(*		nIndexRange[1].nStartIndex := 0;
		nIndexRange[1].nEndIndex := 1;
		nIndexRange[1].bRangeAccess := TRUE; *)
		stNodeAddInfo.nIndexRangeCount := nIndexRangeCount;
		stNodeAddInfo.stIndexRange := stIndexRange;
		iState	:= iState + 1;
	END_IF

1:	(* open UA session *)
	fbUA_Connect(
		Execute				:= TRUE,
		ServerURL			:= sOpcUA_URL,
		SessionConnectInfo	:= SessionConnectInfo,
		Timeout				:= T#5S,
		ConnectionHdl		=> nConnectionHdl
	);

	IF NOT fbUA_Connect.Busy THEN
		fbUA_Connect(Execute := FALSE);

		IF NOT fbUA_Connect.Error THEN
			(* session open *)
			iState := iState + 1;
		ELSE
			bError			:= TRUE;
			nErrorID		:= fbUA_Connect.ErrorID;
			nConnectionHdl	:= 0;
			iState 			:= 0; (* idle *)
		END_IF
	END_IF


2:	(* GetNS Index *)
	fbUA_GetNamespaceIndex(
		Execute			:= TRUE,
		ConnectionHdl	:= nConnectionHdl,
		NamespaceUri	:= 'PLC1',
		NamespaceIndex	=> nNamespaceIndex
	);

	IF NOT fbUA_GetNamespaceIndex.Busy THEN
		fbUA_GetNamespaceIndex(Execute := FALSE);
		IF NOT fbUA_GetNamespaceIndex.Error THEN
			(* session closed *)
			iState 		:= iState + 1; (* idle *)
		ELSE
			bError		:= TRUE;
			nErrorID	:= fbUA_GetNamespaceIndex.ErrorID;
			iState 		:= 6; (* idle *)
		END_IF
	END_IF


3:	(* Get Node Handle *)
	NodeID.eIdentifierType := eUAIdentifierType_String;
	NodeID.nNamespaceIndex := nNamespaceIndex;
	NodeID.sIdentifier	:= 'invalidArrayDef';
	fbUA_NodeGetHandle(
		Execute			:= TRUE,
		ConnectionHdl	:= nConnectionHdl,
		NodeID			:= NodeID,
		NodeHdl			=> nNodeHdl
	);

	IF NOT fbUA_NodeGetHandle.Busy THEN
		fbUA_NodeGetHandle(Execute := FALSE);

		IF NOT fbUA_NodeGetHandle.Error THEN
			(* session closed *)
			iState 					:= iState + 1; (* idle *)
		ELSE
			bError		:= TRUE;
			nErrorID	:= fbUA_NodeGetHandle.ErrorID;
			iState 		:= 6; (* idle *)
			IF fbUA_NodeGetHandle.ErrorID = 16#E4DD0125 THEN  
				bTestSuccessfull := TRUE;
			END_IF

		END_IF
	END_IF


4: 	(* Should not be reached since gethandle should fail! *)
	iState 		:= iState + 1; 
	bTestSuccessfull := FALSE;
	
5:	(* Release Node Handle *)
	fbUA_NodeReleaseHandle(
		Execute			:= TRUE,
		ConnectionHdl	:= nConnectionHdl,
		NodeHdl			:= nNodeHdl
	);

	IF NOT fbUA_NodeReleaseHandle.Busy THEN
		fbUA_NodeReleaseHandle(Execute := FALSE);

		IF NOT fbUA_NodeReleaseHandle.Error THEN
			(* session closed *)
			iState 		:= iState + 1; (* idle *)
		ELSE
			bError		:= TRUE;
			nErrorID	:= fbUA_NodeReleaseHandle.ErrorID;
			iState 		:= 6; (* idle *)
		END_IF
	END_IF


6:	(* close session *)
	fbUA_Disconnect(
		Execute			:= TRUE,
		ConnectionHdl	:= nConnectionHdl
	);

	IF NOT fbUA_Disconnect.Busy THEN
		fbUA_Disconnect(Execute := FALSE);
		bBusy := FALSE;
		IF NOT fbUA_Disconnect.Error THEN
			(* session closed *)
			iState 		:= 0; (* idle *)
			IF NOT bError THEN 
				bDone 	:= TRUE;
			END_IF
		ELSE
			bError			:= TRUE;
			nErrorID		:= fbUA_Disconnect.ErrorID;
			iState 			:= 0; (* idle *)
			nConnectionHdl	:= 0;
		END_IF
	END_IF
END_CASE

END_PROGRAM

// ---- Tests_Henning/POUs/PRG_READ_List_Henning.TcPOU
PROGRAM PRG_READ_List_Henning
VAR
	fbUA_ConnectEx			: UA_ConnectEx;
	SessionConnectInfoEx	: ST_UASessionConnectInfoEx;
	sOpcUA_URL				: STRING(MAX_STRING_LENGTH);
	nConnectionHdl			: DWORD;

	fbUA_GetNamespaceIndex 	: UA_GetNamespaceIndex;
	nNamespaceIndex			: UINT;
	fbUA_NodeGetHandleList	: UA_NodeGetHandleList;
	fbUA_NodeGetHandle		: UA_NodeGetHandle;
	NodeIDCount				: UINT := 2; 
	NodeIDs					: ARRAY [1..nMaxNodeIDsInList] OF ST_UANodeID;
	NodeID1					: ST_UANodeID; 
	NodeID2					: ST_UANodeID; 
	nNodeHdls				: ARRAY [1..nMaxNodeIDsInList] OF DWORD;

	fbUA_ReadList			: UA_ReadList;
	NodeHdlCount			: UINT := 2; 
	stIndexRange			: ARRAY [1..nMaxIndexRange] OF ST_UAIndexRange;
	nIndexRangeCount		: UINT;
	stNodeAddInfo			: ARRAY [1..nMaxNodeIDsInList] OF ST_UANodeAdditionalInfo;
	stReadListData			: ST_ReadListData; // memory block must contain the Data[], NodeErrorIDs[], TimeStamps[] and cbData_R[]
	cbData					: ARRAY [1..nMaxNodeIDsInList] OF UDINT; (* Bytes to be actually Read *)
	cbData_R				: UDINT;
	cbDataTotal				: UDINT; 
	
	fbUA_NodeReleaseHandleList	: UA_NodeReleaseHandleList;

	fbUA_Disconnect		: UA_Disconnect;

	iState		: INT;
	bTest		: BOOL:= TRUE;  
	bDone		: BOOL;
	bBusy		: BOOL;
	bError		: BOOL;
	nErrorID	: DWORD;
END_VAR


CASE iState OF
0:	(* idle *)
	IF bTest THEN
		bTest		:= FALSE;
		bError		:= FALSE;
		nErrorID	:= 0;

		(* Parameterize *)
		sOpcUA_URL						:= 'opc.tcp://henningm-nb:4842';	(* OpcUA Url of the device with ip address *)

		SessionConnectInfoEx.tConnectTimeout 		:= T#5S;
		SessionConnectInfoEx.tSessionTimeout 		:= T#5S;
		SessionConnectInfoEx.sApplicationName		:= '';
		SessionConnectInfoEx.eSecurityMode 			:= eUASecurityMsgMode_None;
		SessionConnectInfoEx.eSecurityPolicyUri 	:= eUASecurityPolicy_None;
		SessionConnectInfoEx.eTransportProfileUri 	:= eUATransportProfileUri_UATcp;
		SessionConnectInfoEx.stUserIdentTokenType.eUserIdentTokenType  	 := eUAUITT_Anonymous; 
		SessionConnectInfoEx.stUserIdentTokenType.sTokenParam1  		 := 'beckhoff\henningm'; 
		SessionConnectInfoEx.stUserIdentTokenType.sTokenParam2  		 := 'xx'; 
		

(*		nIndexRange[1].nStartIndex := 0;
		nIndexRange[1].nEndIndex := 1;
		nIndexRange[1].bRangeAccess := TRUE; *)
		iState	:= iState + 1;
	END_IF

1:	(* open UA session *)
	fbUA_ConnectEx(
		Execute				:= TRUE,
		ServerURL			:= sOpcUA_URL,
		SessionConnectInfoEx:= SessionConnectInfoEx,
		Timeout				:= T#5S,
		ConnectionHdl		=> nConnectionHdl
	);

	IF NOT fbUA_ConnectEx.Busy THEN
		fbUA_ConnectEx(Execute := FALSE);

		IF NOT fbUA_ConnectEx.Error THEN
			(* session open *)
			iState := iState + 1;
		ELSE
			bError			:= TRUE;
			nErrorID		:= fbUA_ConnectEx.ErrorID;
			nConnectionHdl	:= 0;
			iState 			:= 8; (* idle *)
		END_IF
	END_IF


2:	(* GetNS Index *)
	fbUA_GetNamespaceIndex(
		Execute			:= TRUE,
		ConnectionHdl	:= nConnectionHdl,
		NamespaceUri	:= 'urn:HENNINGM-NB:BeckhoffAutomation:Ua:TpyPLC',
		NamespaceIndex	=> nNamespaceIndex
	);

	IF NOT fbUA_GetNamespaceIndex.Busy THEN
		fbUA_GetNamespaceIndex(Execute := FALSE);
		IF NOT fbUA_GetNamespaceIndex.Error THEN
			(* session closed *)
			iState 		:= iState + 1; (* idle *)
		ELSE
			bError		:= TRUE;
			nErrorID	:= fbUA_GetNamespaceIndex.ErrorID;
			iState 		:= 8; (* idle *)
		END_IF
	END_IF


3:	(* Get Node Handle *)
	NodeID1.eIdentifierType := eUAIdentifierType_String;	(* Get Node Handle *)
	NodeID1.nNamespaceIndex := nNamespaceIndex;
	NodeID1.sIdentifier	:= 'MAIN.iVar1';
	fbUA_NodeGetHandle(
		Execute			:= TRUE,
		ConnectionHdl	:= nConnectionHdl,
		NodeID			:= NodeID1,
		NodeHdl			=> nNodeHdls[1]
	);

	IF NOT fbUA_NodeGetHandle.Busy THEN
		fbUA_NodeGetHandle(Execute := FALSE);

		IF NOT fbUA_NodeGetHandle.Error THEN
			(* node handle received successfully *)
			iState 		:= iState + 1; (* UA_Read *)
		ELSE
			bError		:= TRUE;
			nErrorID	:= fbUA_NodeGetHandle.ErrorID;
			iState 		:= 5; (* release node handle *)
		END_IF
	END_IF;

4:	(* Get Node Handle *)
	NodeID2.eIdentifierType := eUAIdentifierType_String;	(* Get Node Handle *)
	NodeID2.nNamespaceIndex := nNamespaceIndex;
	NodeID2.sIdentifier	:= 'MAIN.iVar2';
	fbUA_NodeGetHandle(
		Execute			:= TRUE,
		ConnectionHdl	:= nConnectionHdl,
		NodeID			:= NodeID2,
		NodeHdl			=> nNodeHdls[2]
	);

	IF NOT fbUA_NodeGetHandle.Busy THEN
		fbUA_NodeGetHandle(Execute := FALSE);

		IF NOT fbUA_NodeGetHandle.Error THEN
			(* node handle received successfully *)
			iState 		:= iState + 1; (* UA_Read *)
		ELSE
			bError		:= TRUE;
			nErrorID	:= fbUA_NodeGetHandle.ErrorID;
			iState 		:= 8; (* release node handle *)
		END_IF
	END_IF;
	
5: 	(* UA_Read *)
	cbData[1] := SIZEOF(stReadListData.nIntVar1);
	cbData[2] := SIZEOF(stReadListData.nIntVar2);
	cbDataTotal := SIZEOF(stReadListData);
	fbUA_ReadList(
		Execute			:= TRUE,
		ConnectionHdl	:= nConnectionHdl,
		NodeHdlCount	:= NodeHdlCount, // 2
		NodeHdls		:= nNodeHdls,
		stNodeAddInfo 	:= stNodeAddInfo,
		pVariable		:= ADR(stReadListData),
		cbData			:= cbData ,
		cbDataTotal		:= cbDataTotal		
		);

	IF NOT fbUA_ReadList.Busy THEN
		fbUA_ReadList( Execute := FALSE, cbData_R => cbData_R);

		IF NOT fbUA_ReadList.Error THEN
			(* session closed *)
			iState 		:= iState + 1; (* idle *)
		ELSE
			bError		:= TRUE;
			nErrorID	:= fbUA_ReadList.ErrorID;
			iState 		:= 8; (* idle *)
		END_IF
	END_IF


6:	(* Release Node Handle *)
	fbUA_NodeReleaseHandleList(
		Execute			:= TRUE,
		ConnectionHdl	:= nConnectionHdl,
		NodeHdlCount	:= NodeHdlCount,
		NodeHdls		:= nNodeHdls
	);

	IF NOT fbUA_NodeReleaseHandleList.Busy THEN
		fbUA_NodeReleaseHandleList(Execute := FALSE);

		IF NOT fbUA_NodeReleaseHandleList.Error THEN
			(* session closed *)
			iState 		:= iState + 1; (* idle *)
		ELSE
			bError		:= TRUE;
			nErrorID	:= fbUA_NodeReleaseHandleList.ErrorID;
			iState 		:= 7; (* idle *)
		END_IF
	END_IF


7:	(* close session *)
	fbUA_Disconnect(
		Execute			:= TRUE,
		ConnectionHdl	:= nConnectionHdl
	);

	IF NOT fbUA_Disconnect.Busy THEN
		fbUA_Disconnect(Execute := FALSE);
		bBusy := FALSE;
		IF NOT fbUA_Disconnect.Error THEN
			(* session closed *)
			iState 		:= 0; (* idle *)
			IF NOT bError THEN 
				bDone 	:= TRUE;
			END_IF
		ELSE
			bError			:= TRUE;
			nErrorID		:= fbUA_Disconnect.ErrorID;
			iState 			:= 0; (* idle *)
			nConnectionHdl	:= 0;
		END_IF
	END_IF
END_CASE

END_PROGRAM

// ---- Test_CloudSample/POUs/ADS/FB_CloudAdsSqlInsert.TcPOU
FUNCTION_BLOCK FB_CloudAdsSqlInsert
VAR_INPUT
	sNetID 			: T_AmsNetID	:='';
	sInsertCmd 		: T_MaxString	:='';
	bExecute		: BOOL;
	tTimeout		: TIME 			:= T#15S;
END_VAR
VAR_OUTPUT
	bBusy 			: BOOL;
	bError 			: BOOL;
	nErrID 			: UDINT;
	sSQLState		: ST_DBSQLError := (sSQLState:='',nSQLErrorCode:=0);
END_VAR
VAR
	RisingEdge		: R_TRIG;
	ReturnCode		: UDINT := 0;
	ReturnValues	: ARRAY [0..15] OF BYTE;
	ADSRDWRITE1		: ADSRDWRT;
	state			: BYTE;
	dummy			: ST_internalSQLError;
END_VAR

RisingEdge(CLK:=bExecute);
IF RisingEdge.Q THEN
	state := 1;
END_IF

CASE state OF
	0:
		;
	1:
		bBusy := TRUE;
		bError := FALSE;
		nErrID := 0;

		ReturnCode := 0;
		sSQLState.sSQLState := '';
		sSQLState.nSQLErrorCode := 0;

		MEMSET(ADR(ReturnValues), 0, SIZEOF(ReturnValues));

		ADSRDWRITE1(WRTRD:= FALSE);
		ADSRDWRITE1(
			NETID:= sNetID,
			PORT:= 21372,
			IDXGRP:= 524290,
			IDXOFFS:= 1,
			WRITELEN:= SIZEOF(sInsertCmd),
			SRCADDR:= ADR(sInsertCmd),
			READLEN:= SIZEOF(ReturnValues),
			DESTADDR:= ADR(ReturnValues),
			WRTRD:= TRUE,
			TMOUT:= tTimeout);
		state := 2;
	2:
		ADSRDWRITE1( WRTRD:=FALSE);
		IF NOT ADSRDWRITE1.BUSY THEN
			state:= 3;
		END_IF
	3:
		bBusy := ADSRDWRITE1.BUSY;
		bError := ADSRDWRITE1.ERR;
		nErrID := ADSRDWRITE1.ERRID;

		MEMCPY(ADR(ReturnCode), ADR(ReturnValues)+12, SIZEOF(ReturnCode));

		IF NOT ADSRDWRITE1.ERR THEN
			 IF ReturnCode <> 0 THEN
				bError 	:= TRUE;
				nErrID 	:= ReturnCode;
				MEMCPY(ADR(dummy), ADR(ReturnValues), SIZEOF(dummy));
				sSQLState.nSQLErrorCode := dummy.nSQLErrorCode;
				sSQLState.sSQLState := dummy.sSQLState;
			ELSE
				sSQLState.sSQLState := '00000';
				sSQLState.nSQLErrorCode := 0;
			END_IF
		END_IF
		state := 0;
END_CASE

END_FUNCTION_BLOCK

// ---- Test_CloudSample/POUs/CloudSample.TcPOU
PROGRAM CloudSample
VAR
	(* Declarations for Cloud connect to Microsoft Azure Cloud *)
	bInsertAzure					: BOOL;
	bInsertAzureCyclic				: BOOL;
	nStateAzure						: BYTE := 0;
	R_TRIGAzure						: R_TRIG;
	
	ObjectNodeID					: ST_UANodeID;
	MethodNodeID					: ST_UANodeID;

	bErrorAzure						: BOOL; 
	nErrorIDAzure					: DWORD;
				
	fb_OpcUAConnectAzure			: UA_Connect;
	SessionConnectInfo				: ST_UASessionConnectInfo;
	sOpcUA_URLAzure					: STRING(MAX_STRING_LENGTH);
	hUAConnectionHdlAzure			: UDINT;
	
	fbUA_OpcUAGetNSIndexAzure 		: UA_GetNamespaceIndex;
	nNamespaceIndexAzure			: UINT;
	nNamespaceIndex					: UINT;
	
	fb_OpcUAMethodGetHandleAzure	: UA_MethodGetHandle;
	hUAMethodHandleAzure			: UDINT;
	
	fb_OpcUAMethodCallAzure			: UA_MethodCall;
	hUAMethodCallAzure				: UDINT;
	nUAMethodCallOutputAzure		: ST_UASQLState;
	stOutputArgInfo					: ARRAY [1..nNumberOfOutputArguments] OF ST_UAMethodArgInfo;
	fbBuildSqlInsertAzure			: FB_BuildSQLInsert;
	sSqlInsertAzure					: STRING(100);	
	stOutputArgInfoAndData			: ST_CloudSampleRes;
	
	fb_OpcUADisconnectAzure			: UA_Disconnect;
	bUADisconnectStartAzure			: BOOL; 
	
(* Method Call Struct *)
	InputArguments				: ARRAY [1..nNumberOfInputArguments] OF ST_UAMethodArgInfo; (*ReadWriteReq has 6 input parameters *)
	OutputArguments				: ARRAY [1..1024] OF BYTE; (* Bytes to be read *)
	nArg						: INT;
	nInputData					: ARRAY [1..nInputArgSize] OF BYTE; // (sNetID(24) + Port(2) + IG(4) + IO(4))
	nOffset						: UDINT;

	
	sNetID						: T_AmsNetId := '127.0.0.1.1.1'; 		(* AmsNetId OF the Target *)
	nPort						: INT; 				(* Port number	*)
	nIndexGroup					: DINT;				(* IndexGroup*)
	nIndexOffset				: DINT; 			(* IndexOffset*)
//	cbWriteData					: UDINT;			(* Count of bytes to be read*)
	bInputDataError				: BOOL; 
	
	(* Miscellaneous variables *)
	fbRandom					: DRAND;
	lrRandom					: LREAL;
	sRandom						: STRING(MAX_DATA_ACCURACY);
	sRandom2					: STRING(MAX_DATA_ACCURACY);
	fbNTGetTime					: NT_GetTime;
	bBusyTime					: BOOL;
	stTime						: TIMESTRUCT;
	
	bInit						: BOOL := TRUE;
END_VAR
VAR CONSTANT
	nInputArgSize				: UDINT := 34;  //(sNetID(24) + Port(2) + IG(4) + IO(4))
	nNumberOfInputArguments 	: UDINT := 6;	
	nNumberOfOutputArguments	: UDINT := 1;		(* 6 *)
	cbReadData					: UDINT := SIZEOF(ST_UASQLState);			(* Count of bytes to be read*)
END_VAR

(* Create random number for upload into the Cloud *)
fbRandom(
	Seed := 1,
	Num => lrRandom);
lrRandom := lrRandom * 10;
sRandom := LREAL_TO_STRING(lrRandom);

(* The value of Poti 1 will be used to write into Cloud *)
sRandom2 := INT_TO_STRING(us_Poti_1);
IF bInit THEN 
	M_Init();
	bInit := FALSE; 
END_IF
R_TRIGAzure(CLK := bInsertAzure);
(* Upload once to Microsoft Azure Cloud *)
CASE nStateAzure OF
	0:
	 	(* To start this sample you have to set a rising edge to the variable bInsertAzure *)
		IF R_TRIGAzure.Q OR bInsertAzureCyclic THEN
			M_Init();
			nStateAzure 	:= 1;		
			bInsertAzure 	:= FALSE;
			bInsertAzureCyclic := TRUE;
			bErrorAzure 	:= FALSE; 
			nErrorIDAzure 	:= 0; 
		END_IF
			
	1:
		(* Get System Time to create timestamp*)
		fbNTGetTime(
			NETID 	:= '',
			START	:= TRUE,
			TMOUT 	:= T#5S,
			BUSY 	=> bBusyTime,
			TIMESTR => stTime);
		
		IF NOT bBusyTime THEN
			fbNTGetTime(START := FALSE);
			nStateAzure := 2;
		END_IF

	2:
		(* Establish session to OPC-UA Server *)
		IF hUAConnectionHdlAzure = 0 THEN
			fb_OpcUAConnectAzure(
				Execute 			:= TRUE,
				ServerUrl 			:= 'opc.tcp://ew2013vm.cloudapp.net:4840',
				SessionConnectInfo 	:= SessionConnectInfo,
				Timeout 			:= T#5S,
				ConnectionHdl 		=> hUAConnectionHdlAzure
				);
		ELSE
			nStateAzure := 4; 		
		END_IF
		
		IF NOT fb_OpcUAConnectAzure.Busy THEN
			fb_OpcUAConnectAzure(Execute := FALSE);
			IF NOT fb_OpcUAConnectAzure.Error THEN
				nStateAzure := 3;
			ELSE
				(* Error Occurred *)
				bErrorAzure	 := TRUE; 
				nErrorIDAzure := fb_OpcUAConnectAzure.ErrorID;
			END_IF	
		END_IF	
		
	3: 
		(* GetNS Index *)
		fbUA_OpcUAGetNSIndexAzure(
			Execute			:= TRUE,
			ConnectionHdl	:= hUAConnectionHdlAzure,
			NamespaceUri	:= 'ADSAMS',
			NamespaceIndex	=> nNamespaceIndexAzure
		);
	
		IF NOT fbUA_OpcUAGetNSIndexAzure.Busy THEN
			fbUA_OpcUAGetNSIndexAzure(Execute := FALSE);
			IF NOT fbUA_OpcUAGetNSIndexAzure.Error THEN
				(* session closed *)
				ObjectNodeID.eIdentifierType := eUAIdentifierType_String;
				ObjectNodeID.nNamespaceIndex := nNamespaceIndexAzure;
				ObjectNodeID.sIdentifier	 := 'ADSAMS';
				
				MethodNodeID.eIdentifierType := eUAIdentifierType_String;
				MethodNodeID.nNamespaceIndex := nNamespaceIndexAzure;
				MethodNodeID.sIdentifier	 := 'ADSAMS.AdsReadWriteReq';
				nStateAzure := 4; (* method *)
			ELSE
				(* Error occurred *)
				bErrorAzure	 := TRUE; 
				nErrorIDAzure := fbUA_OpcUAGetNSIndexAzure.ErrorID;
			END_IF
		END_IF
	
	4:
		(* Get method handle for AdsReadWrite method *)
		IF hUAMethodHandleAzure = 0 THEN
			fb_OpcUAMethodGetHandleAzure(
				Execute 		:= TRUE,
				Timeout 		:= T#15S,
				ConnectionHdl  	:= hUAConnectionHdlAzure,
				ObjectNodeID	:= ObjectNodeID,
				MethodNodeID	:= MethodNodeID,
				MethodHdl 		=> hUAMethodHandleAzure);
		END_IF
		
		IF NOT fb_OpcUAMethodGetHandleAzure.Busy THEN 
			fb_OpcUAMethodGetHandleAzure(Execute := FALSE);
			IF NOT fb_OpcUAMethodGetHandleAzure.Error THEN
				nStateAzure := 5;		
			ELSE
				(* Error occurred *)
				bErrorAzure	  := TRUE; 
				nErrorIDAzure := fb_OpcUAMethodGetHandleAzure.ErrorID;
			END_IF
		END_IF 
	
	5:
		(* Prepare SQL Insert for Cloud *)
		fbBuildSqlInsertAzure(
			sTableName 		:= 'Zaehlerdaten',
			stTimestamp 	:= stTime,
			uiMesstellenID 	:= 2,
			stLogger 		:= 'HelloWorld',
			rMesswert 		:= 42,
			stEinheit 		:= 'Celsius',
			sValue 			:= sRandom2,
			sQuery 			=> sSqlInsertAzure);
		
		(* Write data to the Microsoft Azure cloud via OPC-UA *)
		nNamespaceIndex := nNamespaceIndexAzure;
		M_MethodCallInit();
		stOutputArgInfoAndData.stOutputArgInfo[1].nLenData:= SIZEOF(ST_UASQLState);
		IF bInputDataError = FALSE THEN 
			fb_OpcUAMethodCallAzure(
				Execute					:= TRUE,
				Timeout 				:= T#15S,
				ConnectionHdl			:= hUAConnectionHdlAzure,
				MethodHdl				:= hUAMethodHandleAzure,
				nNumberOfInputArguments := nNumberOfInputArguments,		(* 6 *)
				pInputArgInfo			:= ADR(InputArguments),
				cbInputArgInfo			:= SIZEOF(InputArguments),
				pInputArgData			:= ADR(nInputData),
				cbInputArgData			:= nOffset,
				pInputWriteData			:= ADR(sSqlInsertAzure),
				cbInputWriteData		:= INT_TO_UDINT(LEN(sSqlInsertAzure))+1,
				nNumberOfOutputArguments:= nNumberOfOutputArguments,		(* 6 *)
				pOutputArgInfo			:= ADR(stOutputArgInfo),
				cbOutputArgInfo			:= SIZEOF(stOutputArgInfo),
				pOutputArgInfoAndData	:= ADR(stOutputArgInfoAndData),
				cbOutputArgInfoAndData	:= SIZEOF(stOutputArgInfoAndData)		
			);
			IF NOT fb_OpcUAMethodCallAzure.Busy THEN
				fb_OpcUAMethodCallAzure(Execute := FALSE);
				IF NOT fb_OpcUAMethodCallAzure.Error THEN
					bInsertAzure := FALSE;
					nStateAzure := 0;
					nUAMethodCallOutputAzure.nReturnCode := stOutputArgInfoAndData.stUASQLStateInternal.nReturnCode;
					(* ------------ according to TcDatabase.lib *)
					IF nUaMethodCallOutputAzure.nReturnCode <> 0 THEN 
						bErrorAzure := TRUE;
						nErrorIDAzure := stOutputArgInfoAndData.stUASQLStateInternal.nReturnCode;
						nUAMethodCallOutputAzure.sSQLState		:= stOutputArgInfoAndData.stUASQLStateInternal.sSQLState;
						nUAMethodCallOutputAzure.nSQLErrorCode 	:= stOutputArgInfoAndData.stUASQLStateInternal.nSQLErrorCode;
					ELSE
						nUAMethodCallOutputAzure.sSQLState		:= '00000';	
						nUAMethodCallOutputAzure.nSQLErrorCode 	:= 0;		
					END_IF		
					(* ------------- according to TcDatabase.lib *)
				ELSE
					(* Error Occurred *)
					nStateAzure   := 6; 
					bErrorAzure	  := TRUE; 
					nErrorIDAzure := fb_OpcUAMethodCallAzure.ErrorID;
				END_IF	
			END_IF
		ELSE
			(* ERROR nInputData array is too small for the data *)
			(* see M_MethodCallInit*)
			;
		END_IF
END_CASE

ACTION M_Init:
(* Parameterize *)
SessionConnectInfo.tConnectTimeout 		:= T#1S;
SessionConnectInfo.tSessionTimeout 		:= T#1S;
SessionConnectInfo.sApplicationName		:= '';
SessionConnectInfo.sApplicationUri 		:= '';
SessionConnectInfo.eSecurityMode 		:= eUASecurityMsgMode_None;
SessionConnectInfo.eSecurityPolicyUri 	:= eUASecurityPolicy_None;
SessionConnectInfo.eTransportProfileUri := eUATransportProfileUri_UATcp;
END_ACTION

ACTION M_MethodCallInit:
bInputDataError := FALSE; 
(* Method Call parameters *)
sNetID				:= '127.0.0.1.1.1'; 		(* AmsNetId OF the Target *)
nPort				:= 21372; 					(* Port number *) (* AMSPORT_DATABASESRV := 21372 = 16#537C*)
nIndexGroup			:= 16#80002;				(* IndexGroup*) 
nIndexOffset		:= 2; 						(* IndexOffset = DBID (Configurator)*)
//cbWriteData			:= LEN(sSqlInsertAzure)+1;		
//cbReadData			:= 16;	

nOffset := 0;
MEMSET(ADR(InputArguments),0,SIZEOF(InputArguments));
MEMSET(ADR(nInputData),0,SIZEOF(nInputData));

nArg := 1;
(*sNetID := sAmsNetID;*)	(*****l***** NET ID **********)
InputArguments[nArg].DataType			:= eUAType_String;
InputArguments[nArg].ValueRank			:= -1; 							(* Scalar = -1 or Array *)
InputArguments[nArg].ArrayDimensions[1]	:= 0; 							(* Number of Dimension in case its an array *)
InputArguments[nArg].nLenData			:= INT_TO_UDINT(LEN(sNetId)) + 1;				(* Length if its a STRING *)
IF nOffset + INT_TO_UDINT(LEN(sNetId))+1 > nInputArgSize THEN 
	bInputDataError := TRUE;
	RETURN;
ELSE
	MEMCPY(ADR(nInputData)+nOffset,ADR(sNetId),INT_TO_UDINT(LEN(sNetId))+1);				(* VALUE in BYTES FORM *)
	nOffset := nOffset + INT_TO_UDINT(LEN(sNetId))+1;
END_IF

nArg := nArg + 1;
(* nPort := 851;*)			(********** PORT **********)
InputArguments[nArg].DataType			:= eUAType_Int16;
InputArguments[nArg].ValueRank			:= -1; 						(* Scalar = -1 or Array *)
InputArguments[nArg].ArrayDimensions[1]	:= 0; 						(* Number of Dimension in case its an array *)
InputArguments[nArg].nLenData			:= SIZEOF(nPort);			(* Length if its a STRING *)
IF nOffset + SIZEOF(nPort) > nInputArgSize THEN 
	bInputDataError := TRUE;
	RETURN;
ELSE
	MEMCPY(ADR(nInputData)+nOffset,ADR(nPort),SIZEOF(nPort));			(* VALUE in BYTES FORM *)
	nOffset := nOffset + SIZEOF(nPort);
END_IF

nArg := nArg + 1;
(*nIndexGroup := 16#4020;*)	(********** INDEX GROUP **********)
InputArguments[nArg].DataType			:= eUAType_Int32;
InputArguments[nArg].ValueRank			:= -1; 							(* Scalar = -1 or Array *)
InputArguments[nArg].ArrayDimensions[1]	:= 0; 							(* Number of Dimension in case its an array *)
InputArguments[nArg].nLenData			:= SIZEOF(nIndexGroup);			(* Length if its a STRING *)
IF nOffset + SIZEOF(nIndexGroup) > nInputArgSize THEN 
	bInputDataError := TRUE;
	RETURN;
ELSE
	MEMCPY(ADR(nInputData)+nOffset,ADR(nIndexGroup),SIZEOF(nIndexGroup));		(* VALUE in BYTES FORM *)
	nOffset := nOffset + SIZEOF(nIndexGroup);
END_IF


nArg := nArg + 1;
(*nIndexOffset := 0; *)		(********** INDEX OFFSET **********)
InputArguments[nArg].DataType			:= eUAType_Int32;
InputArguments[nArg].ValueRank			:= -1; 							(* Scalar = -1 or Array *)
InputArguments[nArg].ArrayDimensions[1]	:= 0; 							(* Number of Dimension in case its an array *)
InputArguments[nArg].nLenData			:= SIZEOF(nIndexOffset);		(* Length if its a STRING *)
IF nOffset + SIZEOF(nIndexOffset) > nInputArgSize THEN 
	bInputDataError := TRUE;
	RETURN;
ELSE
	MEMCPY(ADR(nInputData)+nOffset,ADR(nIndexOffset),SIZEOF(nIndexOffset));	(* VALUE in BYTES FORM *)
	nOffset := nOffset + SIZEOF(nIndexOffset);
END_IF

nArg := nArg + 1;
(*Data := 2; *)		(*********** WriteData ***********)
InputArguments[nArg].DataType			:= eUAType_ByteString;
InputArguments[nArg].ValueRank			:= -1; 										(* Scalar = -1 or Array *)
InputArguments[nArg].ArrayDimensions[1]	:= 0; 										(* Number of Dimension in case its an array *)
InputArguments[nArg].nLenData			:= INT_TO_UDINT(LEN(sSqlInsertAzure))+1;	(* Length if its a STRING *)

nArg := nArg + 1;
(*Data := 2; *)		(*********** ReadData size ***********)
InputArguments[nArg].DataType			:= eUAType_UInt32;
InputArguments[nArg].ValueRank			:= -1; 						(* Scalar = -1 or Array *)
InputArguments[nArg].ArrayDimensions[1]	:= 0; 						(* Number of Dimension in case its an array *)
InputArguments[nArg].nLenData			:= SIZEOF(cbReadData);		(* Length if its a STRING *)
END_ACTION

END_PROGRAM

// ---- Tests_Henning/POUs/PRG_ArrayTest.TcPOU
PROGRAM PRG_ArrayTest
VAR
	iState: INT;
END_VAR

CASE iState OF
0:	
	PRG_ArrayTest_Read();
	IF(NOT PRG_ArrayTest_Read.bBusy AND NOT PRG_ArrayTest_Read.bError) THEN
		iState := iState+1;
	END_IF
1:
	PRG_ArrayTest_Write();
	IF(NOT PRG_ArrayTest_Write.bBusy AND NOT PRG_ArrayTest_Write.bError) THEN
		iState := iState+1;
	END_IF
2:
	PRG_ArrayTest_ReadWritten();
	IF(NOT PRG_ArrayTest_ReadWritten.bBusy AND NOT PRG_ArrayTest_ReadWritten.bError) THEN
		iState := iState+1;
	END_IF
END_CASE

END_PROGRAM

// ---- Tests_Henning/POUs/PRG_ArrayTest_Read.TcPOU
PROGRAM PRG_ArrayTest_Read
VAR
	fbUA_Connect: UA_Connect;
	SessionConnectInfo: ST_UASessionConnectInfo;
	nConnectionHdl: DWORD;
	fbUA_GetNamespaceIndex: UA_GetNamespaceIndex;
	nNamespaceIndex: UINT;
	fbUA_NodeGetHandle: UA_NodeGetHandle;
	NodeID: ST_UANodeID;
	nNodeHdl: DWORD;
	fbUA_Read: UA_Read;
	stIndexRange: ARRAY[1..nMaxIndexRange] OF ST_UAIndexRange;
	nIndexRangeCount: UINT;
	stNodeAddInfo: ST_UANodeAdditionalInfo;
	Variable: ARRAY[1..nMaxReadData] OF BYTE;
	///DINT; 		// change the data type according to the variable type to be read
	nReadData: STRING;
	fbUA_NodeReleaseHandle: UA_NodeReleaseHandle;
	fbUA_Disconnect: UA_Disconnect;
	iState: INT;
	bTest: BOOL := TRUE;
	bDone: BOOL;
	bBusy: BOOL;
	bError: BOOL;
	nErrorID: DWORD;
	nLoopVars: UINT;
END_VAR

CASE iState OF
0:	(* idle *)
	IF bTest THEN
		bTest		:= FALSE;
		bError		:= FALSE;
		nErrorID	:= 0;
		bBusy 		:= TRUE; 
		SessionConnectInfo.tConnectTimeout 		:= T#9S;
		SessionConnectInfo.tSessionTimeout 		:= T#9S;
		SessionConnectInfo.sApplicationName		:= '';
		SessionConnectInfo.sApplicationUri 		:= '';
		SessionConnectInfo.eSecurityMode 		:= eUASecurityMsgMode_None;
		SessionConnectInfo.eSecurityPolicyUri 	:= eUASecurityPolicy_None;
		SessionConnectInfo.eTransportProfileUri := eUATransportProfileUri_UATcp;

		stNodeAddInfo.nIndexRangeCount := nIndexRangeCount;
		stNodeAddInfo.stIndexRange := stIndexRange;
		iState	:= iState + 1;
	END_IF

1:	(* open UA session *)
	fbUA_Connect(
		Execute				:= TRUE,
		ServerURL			:= GVL_ScalarTests.sOpcUA_URL,
		SessionConnectInfo	:= SessionConnectInfo,
		Timeout				:= T#10S,
		ConnectionHdl		=> nConnectionHdl
	);

	IF NOT fbUA_Connect.Busy THEN
		fbUA_Connect(Execute := FALSE);

		IF NOT fbUA_Connect.Error THEN
			(* session open *)
			iState := iState + 1;
		ELSE
			bError			:= TRUE;
			nErrorID		:= fbUA_Connect.ErrorID;
			nConnectionHdl	:= 0;
			iState 			:= 0; (* idle *)
		END_IF
	END_IF


2:	(* GetNS Index *)
	fbUA_GetNamespaceIndex(
		Execute			:= TRUE,
		ConnectionHdl	:= nConnectionHdl,
		NamespaceUri	:= GVL_ScalarTests.sNodeIDNamespace,
		NamespaceIndex	=> nNamespaceIndex
	);

	IF NOT fbUA_GetNamespaceIndex.Busy THEN
		fbUA_GetNamespaceIndex(Execute := FALSE);

		IF NOT fbUA_GetNamespaceIndex.Error THEN
			(* session closed *)
			iState 		:= iState + 1; (* idle *)
		ELSE
			bError		:= TRUE;
			nErrorID	:= fbUA_GetNamespaceIndex.ErrorID;
			iState 		:= 6; (* idle *)
		END_IF
	END_IF


3:	(* Get Node Handle *)
	NodeID.eIdentifierType := eUAIdentifierType_String;
	NodeID.nNamespaceIndex := nNamespaceIndex;
	NodeID.sIdentifier	:= GVL_ArrayTests.NodeID_Identifiers[nLoopVars]; // 'GVL_static.stat_BSTR_0';
	fbUA_NodeGetHandle(
		Execute			:= TRUE,
		ConnectionHdl	:= nConnectionHdl,
		NodeID			:= NodeID,
		NodeHdl			=> nNodeHdl
	);

	IF NOT fbUA_NodeGetHandle.Busy THEN
		fbUA_NodeGetHandle(Execute := FALSE);

		IF NOT fbUA_NodeGetHandle.Error THEN
			(* session closed *)
			iState 		:= iState + 1; (* idle *)
		ELSE
			bError		:= TRUE;
			nErrorID	:= fbUA_NodeGetHandle.ErrorID;
			iState 		:= 6; (* idle *)
		END_IF
	END_IF


4: 	(* UA_Read *)
	fbUA_Read(
		Execute			:= TRUE,
		ConnectionHdl	:= nConnectionHdl,
		NodeHdl			:= nNodeHdl,
		stNodeAddInfo 	:= stNodeAddInfo,
		cbData			:= GVL_ArrayTests.NodeID_Sizes[nLoopVars], //SIZEOF(nReadData),
		pVariable		:= ADR(GVL_ArrayTests.NodeID_ReadResults[nLoopVars].nData) //Variable
		);

	IF NOT fbUA_Read.Busy THEN
		fbUA_Read(
			Execute 	:= FALSE);

		IF NOT fbUA_Read.Error THEN
			(* session closed *)
			iState 		:= iState + 1; (* idle *)
			//Do we need this? We simply store in UNION! MEMCPY(ADR(nReadData),ADR(Variable),SIZEOF(nReadData));
		ELSE
			bError		:= TRUE;
			nErrorID	:= fbUA_Read.ErrorID;
			iState 		:= 7; (* idle *)
		END_IF
	END_IF



5:	(* Release Node Handle *)
	fbUA_NodeReleaseHandle(
		Execute			:= TRUE,
		ConnectionHdl	:= nConnectionHdl,
		NodeHdl			:= nNodeHdl
	);

	IF NOT fbUA_NodeReleaseHandle.Busy THEN
		fbUA_NodeReleaseHandle(Execute := FALSE);

		IF NOT fbUA_NodeReleaseHandle.Error THEN
			(* session closed *)
			iState 		:= iState + 1; (* idle *)
		ELSE
			bError		:= TRUE;
			nErrorID	:= fbUA_NodeReleaseHandle.ErrorID;
			iState 		:= 6; (* idle *)
		END_IF
	END_IF


6:	(* close session *)
	fbUA_Disconnect(
		Execute			:= TRUE,
		ConnectionHdl	:= nConnectionHdl
	);

	IF NOT fbUA_Disconnect.Busy THEN
		fbUA_Disconnect(Execute := FALSE);

		IF NOT fbUA_Disconnect.Error THEN
			(* session closed *)
			iState 		:= 0; (* idle *)
			//restart with next var, if existing in array
			IF(nLoopVars < nEndOfNodeIDVars) THEN
				nLoopVars := nLoopVars+1;
				bTest := TRUE;
			ELSE 
				bBusy 		:= FALSE;
				//prepare for next call 
				bTest := TRUE;
				nLoopVars := 0;
			END_IF
		ELSE
			bError			:= TRUE;
			nErrorID		:= fbUA_Disconnect.ErrorID;
			iState 			:= 0; (* idle *)
			nConnectionHdl	:= 0;
		END_IF
	END_IF
END_CASE

END_PROGRAM

// ---- Tests_Henning/POUs/PRG_ArrayTest_Write.TcPOU
PROGRAM PRG_ArrayTest_Write
VAR
	fbUA_Connect: UA_Connect;
	SessionConnectInfo: ST_UASessionConnectInfo;
	sOpcUA_URL: STRING(MAX_STRING_LENGTH);
	nConnectionHdl: DWORD;
	fbUA_GetNamespaceIndex: UA_GetNamespaceIndex;
	sNamespaceUri: STRING(MAX_STRING_LENGTH);
	nNamespaceIndex: UINT;
	fbUA_NodeGetHandle: UA_NodeGetHandle;
	NodeID: ST_UANodeID;
	nNodeHdl: DWORD;
	fbUA_Write: UA_Write;
	stIndexRange: ARRAY[1..nMaxIndexRange] OF ST_UAIndexRange;
	nIndexRangeCount: UINT;
	stNodeAddInfo: ST_UANodeAdditionalInfo;
	/// UDINT := 12312345;		// change according to the type of variable
	nWriteData: STRING := 'Hallo';
	Variable: ARRAY[1..nMaxReadData] OF BYTE;
	cbData: UDINT;
	fbUA_NodeReleaseHandle: UA_NodeReleaseHandle;
	fbUA_Disconnect: UA_Disconnect;
	iState: INT;
	bTest: BOOL := TRUE;
	bDone: BOOL;
	bBusy: BOOL;
	bError: BOOL;
	nErrorID: DWORD;
	nLoopVars: UINT;
END_VAR

CASE iState OF
0:	(* idle *)
	IF bTest THEN
		bTest	:= FALSE;
		bError	:= FALSE;
		nErrorID	:= 0;
		bBusy := TRUE; 

		(* Parameterize 
		GVL_ScalarTests.NodeID_WriteCommands[0].bBool := TRUE; 
		GVL_ScalarTests.NodeID_WriteCommands[1].sString := 'WriteTest'; 
		GVL_ScalarTests.NodeID_WriteCommands[2].bByte := 123; 
		GVL_ScalarTests.NodeID_WriteCommands[3].nInt := 124; 
		GVL_ScalarTests.NodeID_WriteCommands[4].nUdint := 125; 
		GVL_ScalarTests.NodeID_WriteCommands[5].nLReal := 1.23456; //R8x 
		GVL_ScalarTests.NodeID_WriteCommands[6].bByte := 111; 
		GVL_ScalarTests.NodeID_WriteCommands[7].nInt := 112; 
		GVL_ScalarTests.NodeID_WriteCommands[8].nUdint := 113; 
		*)
		
		SessionConnectInfo.tConnectTimeout 		:= T#9S;
		SessionConnectInfo.tSessionTimeout 		:= T#9S;
		SessionConnectInfo.sApplicationName		:= '';
		SessionConnectInfo.sApplicationUri 		:= '';
		SessionConnectInfo.eSecurityMode 		:= eUASecurityMsgMode_None;
		SessionConnectInfo.eSecurityPolicyUri 	:= eUASecurityPolicy_None;
		SessionConnectInfo.eTransportProfileUri := eUATransportProfileUri_UATcp;
		
		stNodeAddInfo.nIndexRangeCount := nIndexRangeCount;
		stNodeAddInfo.stIndexRange := stIndexRange;
		iState	:= iState + 1;
	END_IF

1:	(* open UA session *)
	fbUA_Connect(
		Execute				:= TRUE,
		ServerURL			:= GVL_ScalarTests.sOpcUA_URL,
		SessionConnectInfo	:= SessionConnectInfo,
		Timeout				:= T#10S,
		ConnectionHdl		=> nConnectionHdl
	);

	IF NOT fbUA_Connect.Busy THEN
		fbUA_Connect(Execute := FALSE);

		IF NOT fbUA_Connect.Error THEN
			(* session open *)
			iState := iState + 1;
		ELSE
			bError			:= TRUE;
			nErrorID		:= fbUA_Connect.ErrorID;
			nConnectionHdl	:= 0;
			iState 			:= 0; (* idle *)
		END_IF
	END_IF


2:	(* GetNS Index *)
	fbUA_GetNamespaceIndex(
		Execute			:= TRUE,
		ConnectionHdl	:= nConnectionHdl,
		NamespaceUri	:= GVL_ScalarTests.sNodeIDNamespace,
		NamespaceIndex	=> nNamespaceIndex
	);

	IF NOT fbUA_GetNamespaceIndex.Busy THEN
		fbUA_GetNamespaceIndex(Execute := FALSE);

		IF NOT fbUA_GetNamespaceIndex.Error THEN
			(* session closed *)
			iState 		:= iState + 1; (* idle *)
		ELSE
			bError		:= TRUE;
			nErrorID	:= fbUA_GetNamespaceIndex.ErrorID;
			iState 		:= 6; (* idle *)
		END_IF
	END_IF


3:	(* Get Node Handle *)
	NodeID.eIdentifierType := eUAIdentifierType_String;
	NodeID.nNamespaceIndex := nNamespaceIndex;
	NodeID.sIdentifier	:= GVL_ArrayTests.NodeID_Identifiers[nLoopVars]; // 'GVL_static.stat_BSTR_0';
	fbUA_NodeGetHandle(
		Execute			:= TRUE,
		ConnectionHdl	:= nConnectionHdl,
		NodeID			:= NodeID,
		NodeHdl			=> nNodeHdl
	);

	IF NOT fbUA_NodeGetHandle.Busy THEN
		fbUA_NodeGetHandle(Execute := FALSE);

		IF NOT fbUA_NodeGetHandle.Error THEN
			(* session closed *)
			IF SIZEOF(nWriteData) <= nMaxReadData THEN 
				iState 		:= iState + 1; (* idle *)
				MEMSET(ADR(Variable),0,SIZEOF(Variable));
				MEMCPY(ADR(Variable),ADR(nWriteData),SIZEOF(nWriteData));
			ELSE
				//cannot write buffer too small -> increase the value of nMaxData in GVL
				bError		:= TRUE;
				iState 		:= 6; (* idle *)
			END_IF
		ELSE
			bError		:= TRUE;
			nErrorID	:= fbUA_NodeGetHandle.ErrorID;
			iState 		:= 6; (* idle *)
		END_IF
	END_IF


4: 	(* UA_Write *)
	fbUA_Write(
		Execute			:= TRUE,
		ConnectionHdl	:= nConnectionHdl,
		NodeHdl			:= nNodeHdl,
		stNodeAddInfo	:= stNodeAddInfo,
		cbData			:= GVL_ArrayTests.NodeID_Sizes[nLoopVars], //SIZEOF(nWriteData),
		pVariable		:= ADR(GVL_ArrayTests.NodeID_WriteCommands[nLoopVars].nData) // Variable		:= Variable
		);

	IF NOT fbUA_Write.Busy THEN
		fbUA_Write(
			Execute 		:= FALSE);

		IF NOT fbUA_Write.Error THEN
			(* session closed *)
			iState 		:= iState + 1; (* idle *)
		ELSE
			bError		:= TRUE;
			nErrorID	:= fbUA_Write.ErrorID;
			iState 		:= 7; (* idle *)
		END_IF
	END_IF


5:	(* Release Node Handle *)
	fbUA_NodeReleaseHandle(
		Execute			:= TRUE,
		ConnectionHdl	:= nConnectionHdl,
		NodeHdl			:= nNodeHdl
	);

	IF NOT fbUA_NodeReleaseHandle.Busy THEN
		fbUA_NodeReleaseHandle(Execute := FALSE);

		IF NOT fbUA_NodeReleaseHandle.Error THEN
			(* session closed *)
			iState 		:= iState + 1; (* idle *)
		ELSE
			bError		:= TRUE;
			nErrorID	:= fbUA_NodeReleaseHandle.ErrorID;
			iState 		:= 6; (* idle *)
		END_IF
	END_IF


6:	(* close session *)
	fbUA_Disconnect(
		Execute			:= TRUE,
		ConnectionHdl	:= nConnectionHdl
	);

	IF NOT fbUA_Disconnect.Busy THEN
		fbUA_Disconnect(Execute := FALSE);

		IF NOT fbUA_Disconnect.Error THEN
			(* session closed *)
			iState 		:= 0; (* idle *)			//restart with next var, if existing in array
			IF(nLoopVars < nEndOfNodeIDVars) THEN
				nLoopVars := nLoopVars+1;
				bTest := TRUE;
			ELSE 
				bBusy 		:= FALSE;
				//prepare for next call 
				nLoopVars := 0;
			END_IF
		ELSE
			bError		:= TRUE;
			nErrorID	:= fbUA_Disconnect.ErrorID;
			iState 		:= 0; (* idle *)
			nConnectionHdl	:= 0;
		END_IF
	END_IF
END_CASE

END_PROGRAM

// ---- Tests_Henning/POUs/PRG_ArrayTest_ReadWritten.TcPOU
PROGRAM PRG_ArrayTest_ReadWritten
VAR
	fbUA_Connect: UA_Connect;
	SessionConnectInfo: ST_UASessionConnectInfo;
	nConnectionHdl: DWORD;
	fbUA_GetNamespaceIndex: UA_GetNamespaceIndex;
	nNamespaceIndex: UINT;
	fbUA_NodeGetHandle: UA_NodeGetHandle;
	NodeID: ST_UANodeID;
	nNodeHdl: DWORD;
	fbUA_Read: UA_Read;
	stIndexRange: ARRAY[1..nMaxIndexRange] OF ST_UAIndexRange;
	nIndexRangeCount: UINT;
	stNodeAddInfo: ST_UANodeAdditionalInfo;
	Variable: ARRAY[1..nMaxReadData] OF BYTE;
	///DINT; 		// change the data type according to the variable type to be read
	nReadData: STRING;
	fbUA_NodeReleaseHandle: UA_NodeReleaseHandle;
	fbUA_Disconnect: UA_Disconnect;
	iState: INT;
	bTest: BOOL := TRUE;
	bDone: BOOL;
	bBusy: BOOL;
	bError: BOOL;
	nErrorID: DWORD;
	nLoopVars: UINT;
	counter: UDINT;
	a: ARRAY[1..nMaxReadDataArray] OF BYTE;
	b: ARRAY[1..nMaxReadDataArray] OF BYTE;
	a_: BYTE;
	b_: BYTE;
	nTmpL: UINT;
END_VAR

CASE iState OF
0:	(* idle *)
	IF bTest THEN
		bTest		:= FALSE;
		bError		:= FALSE;
		nErrorID	:= 0;
		bBusy 		:= TRUE; 
		SessionConnectInfo.tConnectTimeout 		:= T#9S;
		SessionConnectInfo.tSessionTimeout 		:= T#9S;
		SessionConnectInfo.sApplicationName		:= '';
		SessionConnectInfo.sApplicationUri 		:= '';
		SessionConnectInfo.eSecurityMode 		:= eUASecurityMsgMode_None;
		SessionConnectInfo.eSecurityPolicyUri 	:= eUASecurityPolicy_None;
		SessionConnectInfo.eTransportProfileUri := eUATransportProfileUri_UATcp;

		stNodeAddInfo.nIndexRangeCount := nIndexRangeCount;
		stNodeAddInfo.stIndexRange := stIndexRange;
		iState	:= iState + 1;
	END_IF

1:	(* open UA session *)
	fbUA_Connect(
		Execute				:= TRUE,
		ServerURL			:= GVL_ScalarTests.sOpcUA_URL,
		SessionConnectInfo	:= SessionConnectInfo,
		Timeout				:= T#10S,
		ConnectionHdl		=> nConnectionHdl
	);

	IF NOT fbUA_Connect.Busy THEN
		fbUA_Connect(Execute := FALSE);

		IF NOT fbUA_Connect.Error THEN
			(* session open *)
			iState := iState + 1;
		ELSE
			bError			:= TRUE;
			nErrorID		:= fbUA_Connect.ErrorID;
			nConnectionHdl	:= 0;
			iState 			:= 0; (* idle *)
		END_IF
	END_IF


2:	(* GetNS Index *)
	fbUA_GetNamespaceIndex(
		Execute			:= TRUE,
		ConnectionHdl	:= nConnectionHdl,
		NamespaceUri	:= GVL_ScalarTests.sNodeIDNamespace,
		NamespaceIndex	=> nNamespaceIndex
	);

	IF NOT fbUA_GetNamespaceIndex.Busy THEN
		fbUA_GetNamespaceIndex(Execute := FALSE);

		IF NOT fbUA_GetNamespaceIndex.Error THEN
			(* session closed *)
			iState 		:= iState + 1; (* idle *)
		ELSE
			bError		:= TRUE;
			nErrorID	:= fbUA_GetNamespaceIndex.ErrorID;
			iState 		:= 6; (* idle *)
		END_IF
	END_IF


3:	(* Get Node Handle *)
	NodeID.eIdentifierType := eUAIdentifierType_String;
	NodeID.nNamespaceIndex := nNamespaceIndex;
	NodeID.sIdentifier	:= GVL_ArrayTests.NodeID_Identifiers[nLoopVars]; // 'GVL_static.stat_BSTR_0';
	fbUA_NodeGetHandle(
		Execute			:= TRUE,
		ConnectionHdl	:= nConnectionHdl,
		NodeID			:= NodeID,
		NodeHdl			=> nNodeHdl
	);

	IF NOT fbUA_NodeGetHandle.Busy THEN
		fbUA_NodeGetHandle(Execute := FALSE);

		IF NOT fbUA_NodeGetHandle.Error THEN
			(* session closed *)
			iState 		:= iState + 1; (* idle *)
		ELSE
			bError		:= TRUE;
			nErrorID	:= fbUA_NodeGetHandle.ErrorID;
			iState 		:= 6; (* idle *)
		END_IF
	END_IF


4: 	(* UA_Read *)
	fbUA_Read(
		Execute			:= TRUE,
		ConnectionHdl	:= nConnectionHdl,
		NodeHdl			:= nNodeHdl,
		stNodeAddInfo 	:= stNodeAddInfo,
		cbData			:= GVL_ArrayTests.NodeID_Sizes[nLoopVars], //SIZEOF(nReadData),		
		pVariable		:= ADR(GVL_ArrayTests.NodeID_ReadWrittenResults[nLoopVars].nData) //Variable
		);

	IF NOT fbUA_Read.Busy THEN
		fbUA_Read(
			Execute 	:= FALSE);

		IF NOT fbUA_Read.Error THEN
			(* session closed *)
			iState 		:= iState + 1; (* idle *)
			a := GVL_ArrayTests.NodeID_WriteCommands[nLoopVars].nData;
			b := GVL_ArrayTests.NodeID_ReadWrittenResults[nLoopVars].nData;
			FOR counter:=1 TO fbUA_Read.cbData_R //fbUA_Read.GVL_ScalarTests.NodeID_Sizes[nLoopVars]
			DO
				a_ := a[counter];
				b_ := b[counter];
				IF(NOT a_ = b_) THEN
					EXIT;
				END_IF
			END_FOR
			IF(Counter = fbUA_Read.cbData_R+1) THEN //GVL_ScalarTests.NodeID_Sizes[nLoopVars]+1) THEN //all bytes are equal as long as length site is defined
				GVL_ArrayTests.NodeID_CheckReadWrite[nLoopVars] := TRUE;
			END_IF 
			//Do we need this? We simply store in UNION! MEMCPY(ADR(nReadData),ADR(Variable),SIZEOF(nReadData));
		ELSE
			bError		:= TRUE;
			nErrorID	:= fbUA_Read.ErrorID;
			iState 		:= 7; (* idle *)
		END_IF
	END_IF



5:	(* Release Node Handle *)
	fbUA_NodeReleaseHandle(
		Execute			:= TRUE,
		ConnectionHdl	:= nConnectionHdl,
		NodeHdl			:= nNodeHdl
	);

	IF NOT fbUA_NodeReleaseHandle.Busy THEN
		fbUA_NodeReleaseHandle(Execute := FALSE);

		IF NOT fbUA_NodeReleaseHandle.Error THEN
			(* session closed *)
			iState 		:= iState + 1; (* idle *)
		ELSE
			bError		:= TRUE;
			nErrorID	:= fbUA_NodeReleaseHandle.ErrorID;
			iState 		:= 6; (* idle *)
		END_IF
	END_IF


6:	(* close session *)
	fbUA_Disconnect(
		Execute			:= TRUE,
		ConnectionHdl	:= nConnectionHdl
	);

	IF NOT fbUA_Disconnect.Busy THEN
		fbUA_Disconnect(Execute := FALSE);

		IF NOT fbUA_Disconnect.Error THEN
			(* session closed *)
			iState 		:= 0; (* idle *)
			//restart with next var, if existing in array
			IF(nLoopVars < nEndOfNodeIDVars) THEN
				nLoopVars := nLoopVars+1;
				bTest := TRUE;
			ELSE 
				bBusy 		:= FALSE;
				//prepare for next call 
				bTest := TRUE;
				nLoopVars := 0;
			END_IF
		ELSE
			bError			:= TRUE;
			nErrorID		:= fbUA_Disconnect.ErrorID;
			iState 			:= 0; (* idle *)
			nConnectionHdl	:= 0;
		END_IF
	END_IF
END_CASE

END_PROGRAM

// ---- Tests_Henning/POUs/PRG_CallInOut1DimParam.TcPOU
PROGRAM PRG_CallInOut1DimParam
VAR
	///CallInOutMultiParams(numberIn1(uInt32),numberIn2(UInt32),numberOut1(UInt32),numberOut2(UINT32));
	fbUA_Connect		: UA_Connect;
	SessionConnectInfo	: ST_UASessionConnectInfo;
	sOpcUA_URL			: STRING(MAX_STRING_LENGTH);
	nConnectionHdl		: DWORD;
	
	fbUA_GetNamespaceIndex	: UA_GetNamespaceIndex;
	nNamespaceIndex			: UINT;
	
	fbUA_MethodGetHandle: UA_MethodGetHandle;
	nMethodHdl			: DWORD;
	ObjectNodeID		: ST_UANodeID;
	MethodNodeID		: ST_UANodeID;
	fbUA_MethodCall		: UA_MethodCall;
	InputArguments		: ARRAY[1..nNumberOfInputArguments] OF ST_UAMethodArgInfo;
	nInputData			: ARRAY[1..nInputArgSize] OF BYTE;
	stOutputArgInfoAndData	: ST_UAMethodCall_CallInOut1DimParam;
	stOutputArgInfo		: ARRAY[1..nNumberOfOutputArguments] OF ST_UAMethodArgInfo;
	numberIn1			: UDINT;
	numberIn2			: UDINT;
	
	fbUA_MethodReleaseHandle	: UA_MethodReleaseHandle;
	
	fbUA_Disconnect	: UA_Disconnect;
	
	/// Count of bytes to be written 
	cbWriteData		: UDINT;
	
	nArg			: INT;
	nOffset			: UDINT;
	bInputDataError	: BOOL;
	bTest			: BOOL := TRUE;
	bDone			: BOOL;
	bBusy			: BOOL;
	bError			: BOOL;
	nErrorID		: DWORD;
	iState			: INT;
	
END_VAR
VAR CONSTANT
	nNumberOfInputArguments	: UDINT := 1;
	nNumberOfOutputArguments: UDINT := 1;
	nInputArgSize			: UDINT := 8; 
END_VAR

(*
CallInOut1DimParams(	[numberIn1(uInt32),	numberIn2(UInt32)]
						[numberOut1(UInt32),numberOut2(UINT32),	numberOut3(UINT32)]
);
*)

CASE iState OF

0:	(* idle *)
	IF bTest THEN
		bTest		:= FALSE;
		bError		:= FALSE;
		nErrorID	:= 0;
		stOutputArgInfoAndData.output1 	:= 0; 
		stOutputArgInfoAndData.output2 	:= 0; 
		stOutputArgInfoAndData.output3 	:= 0; 
		(* Parameterize *)
		sOpcUA_URL		:= 'opc.tcp://localhost:4841';	(* OpcUA Url of the device with ip address *)

		SessionConnectInfo.tConnectTimeout 		:= T#9M;
		SessionConnectInfo.tSessionTimeout 		:= T#9M;
		SessionConnectInfo.sApplicationName		:= '';
		SessionConnectInfo.sApplicationUri 		:= '';
		SessionConnectInfo.eSecurityMode 		:= eUASecurityMsgMode_None;
		SessionConnectInfo.eSecurityPolicyUri 	:= eUASecurityPolicy_None;
		SessionConnectInfo.eTransportProfileUri := eUATransportProfileUri_UATcp;

		iState	:= iState + 1;
	END_IF

1:	(* open UA session *)
	fbUA_Connect(
		Execute				:= TRUE,
		ServerURL			:= sOpcUA_URL,
		SessionConnectInfo	:= SessionConnectInfo,
		Timeout				:= T#10S,
		ConnectionHdl		=> nConnectionHdl
	);

	IF NOT fbUA_Connect.Busy THEN
		fbUA_Connect(Execute := FALSE);

		IF NOT fbUA_Connect.Error THEN
			(* connected *)
			iState := iState + 1;
		ELSE
			bError			:= TRUE;
			nErrorID		:= fbUA_Connect.ErrorID;
			nConnectionHdl	:= 0;
			iState 			:= 0; (* idle *)
		END_IF
	END_IF


2:	(* GetNS Index *)
	fbUA_GetNamespaceIndex(
		Execute			:= TRUE,
		ConnectionHdl	:= nConnectionHdl,
		NamespaceUri	:= 'PLC1',
		NamespaceIndex	=> nNamespaceIndex
	);

	IF NOT fbUA_GetNamespaceIndex.Busy THEN
		fbUA_GetNamespaceIndex(Execute := FALSE);

		IF NOT fbUA_GetNamespaceIndex.Error THEN
			(* namespace index read successfully *)
			iState 		:= iState + 1; (* get node handle *)
		ELSE
			bError		:= TRUE;
			nErrorID	:= fbUA_GetNamespaceIndex.ErrorID;
			iState 		:= 7; (* disconnect *)
		END_IF
	END_IF

3:	(* Get Method Handle *)
		ObjectNodeID.eIdentifierType := eUAIdentifierType_String;
		ObjectNodeID.nNamespaceIndex := nNamespaceIndex;
		ObjectNodeID.sIdentifier	:= 'TestMethods';
	
		MethodNodeID.eIdentifierType := eUAIdentifierType_String;
		MethodNodeID.nNamespaceIndex := nNamespaceIndex;
		MethodNodeID.sIdentifier	:= 'TestMethods.CallInOut1DimParam';

		M_Init();
		IF bInputDataError = FALSE THEN
			iState 	:= iState + 1;
		ELSE
			bBusy		:= FALSE; 
			bError 		:= TRUE;
			nErrorID 	:= 16#70A; //out of memory
		END_IF


4:	(* Method Get Handle *)
	fbUA_MethodGetHandle(
			Execute			:= TRUE,
			ConnectionHdl	:= nConnectionHdl,
			ObjectNodeID	:= ObjectNodeID,
			MethodNodeID 	:= MethodNodeID,
			MethodHdl		=> nMethodHdl
		);
	IF NOT fbUA_MethodGetHandle.Busy THEN
		fbUA_MethodGetHandle(Execute := FALSE);

		IF NOT fbUA_MethodGetHandle.Error THEN
			(*  *)
			iState := iState + 1; (* Call Method *)
		ELSE
			bError		:= TRUE;
			nErrorID	:= fbUA_MethodGetHandle.ErrorID;
			iState	 	:= 6; (* Release method Handle *)
		END_IF
	END_IF


5:	(* Method Call *)
	fbUA_MethodCall(
		Execute					:= TRUE,
		Timeout					:= T#20S,
		ConnectionHdl			:= nConnectionHdl,
		MethodHdl				:= nMethodHdl,
		nNumberOfInputArguments := nNumberOfInputArguments, 
		pInputArgData			:= ADR(nInputData),
		cbInputArgData			:= cbWriteData,
		pInputArgInfo			:= ADR(InputArguments),
		cbInputArgInfo			:= SIZEOF(InputArguments),
		nNumberOfOutputArguments:= nNumberOfOutputArguments,
		pOutputArgInfo			:= ADR(stOutputArgInfo),
		cbOutputArgInfo			:= SIZEOF(stOutputArgInfo),
		pOutputArgInfoAndData	:= ADR(stOutputArgInfoAndData),
		cbOutputArgInfoAndData	:= SIZEOF(stOutputArgInfoAndData)	
	);
	IF NOT fbUA_MethodCall.Busy THEN
		fbUA_MethodCall(Execute := FALSE);
		IF NOT fbUA_MethodCall.Error THEN
			(*  *)
			iState 	:= iState + 1; (* Release handle *)
		ELSE
			bError		:= TRUE;
			nErrorID	:= fbUA_MethodCall.ErrorID;
			iState		:= 6; (* Release method handle *)
		END_IF
	END_IF


6:	(* Release Method Handle *)
	fbUA_MethodReleaseHandle(
		Execute			:= TRUE,
		ConnectionHdl	:= nConnectionHdl,
		MethodHdl		:= nMethodHdl
	);

	IF NOT fbUA_MethodReleaseHandle.Busy THEN
		fbUA_MethodReleaseHandle(Execute := FALSE);
		bBusy := FALSE;
		IF NOT fbUA_MethodReleaseHandle.Error THEN
			(* session closed *)
			iState 	:= 7; (* Disconnect *)
		ELSE
			bError		:= TRUE;
			nErrorID	:= fbUA_MethodReleaseHandle.ErrorID;
			iState 		:= 7; (* Disconnect *)
		END_IF
	END_IF
	
7:	(* Disconnect *) 
	fbUA_Disconnect(
		Execute			:= TRUE,
		ConnectionHdl	:= nConnectionHdl
	);

	IF NOT fbUA_Disconnect.Busy THEN
		fbUA_Disconnect(Execute := FALSE);

		IF NOT fbUA_Disconnect.Error THEN
			(* disconnected *)
			iState 	:= 0; (* idle *)
			bDone 	:= TRUE;
			bBusy 	:= FALSE;
		ELSE
			bBusy 			:= FALSE;
			bError			:= TRUE;
			nErrorID		:= fbUA_Disconnect.ErrorID;
			iState 			:= 0; (* idle *)
			nConnectionHdl	:= 0;
		END_IF
	END_IF
END_CASE

ACTION M_Init:
bInputDataError := FALSE; 
nOffset := 0;
MEMSET(ADR(InputArguments),0,SIZEOF(InputArguments));
MEMSET(ADR(nInputData),0,SIZEOF(nInputData));

nArg := 1;
(*numberIn1*)			(********** Input parameter 1 **********)
InputArguments[nArg].DataType			:= eUAType_UInt32;
InputArguments[nArg].ValueRank			:= 1; 							(* Scalar = -1 or 1Dim-Array =1*)
InputArguments[nArg].ArrayDimensions[1]	:= 2; 							(* Number of Dimension in case its an array *)
InputArguments[nArg].nLenData			:= SIZEOF(numberIn1)+SIZEOF(numberIn2);			(* Length if its a STRING *)

IF nOffset + SIZEOF(numberIn1)+SIZEOF(numberIn2) > nInputArgSize THEN 
	bInputDataError := TRUE;
	RETURN;
ELSE
	MEMCPY(ADR(nInputData)+nOffset,ADR(numberIn1),SIZEOF(numberIn1));				(* VALUE in BYTES FORM *)
	nOffset := nOffset + SIZEOF(numberIn1);
	MEMCPY(ADR(nInputData)+nOffset,ADR(numberIn2),SIZEOF(numberIn2));				(* VALUE in BYTES FORM *)
	nOffset := nOffset + SIZEOF(numberIn2);
END_IF
cbWriteData := nOffset;

//************** Prepare Output Argument information ***********
stOutputArgInfo[1].nLenData := 	SIZEOF(stOutputArgInfoAndData.output1) +
								SIZEOF(stOutputArgInfoAndData.output2) +
								SIZEOF(stOutputArgInfoAndData.output3);
END_ACTION

END_PROGRAM

// ---- Tests_Henning/POUs/PRG_CallInOut1DimStringParam.TcPOU
PROGRAM PRG_CallInOut1DimStringParam
VAR
	///CallInOutMultiParams(numberIn1(uInt32),numberIn2(UInt32),numberOut1(UInt32),numberOut2(UINT32));
	//sIn1: STRING := 'Hallooooo';
	//sIn2: STRING := 'test';
	fbUA_Connect		: UA_Connect;
	SessionConnectInfo	: ST_UASessionConnectInfo;
	sOpcUA_URL			: STRING(MAX_STRING_LENGTH);
	nConnectionHdl		: DWORD;
	
	fbUA_GetNamespaceIndex	: UA_GetNamespaceIndex;
	nNamespaceIndex			: UINT;
	
	fbUA_MethodGetHandle: UA_MethodGetHandle;
	nMethodHdl			: DWORD;
	ObjectNodeID		: ST_UANodeID;
	MethodNodeID		: ST_UANodeID;
	
	fbUA_MethodCall		: UA_MethodCall;
	InputArguments		: ARRAY[1..nNumberOfInputArguments] OF ST_UAMethodArgInfo;
	sInArray			: ARRAY[1..2] OF STRING := ['Halloooo', 'test'] ;
	stOutputArgInfoAndData	: ST_UAMethodCall_CallInOut1DimStringParam;
	nInputData			: ARRAY[1..nInputArgSize] OF BYTE;
	stOutputArgInfo 	: ARRAY[1..nNumberOfOutputArguments] OF ST_UAMethodArgInfo;
	
	fbUA_MethodReleaseHandle: UA_MethodReleaseHandle;
	
	fbUA_Disconnect			: UA_Disconnect;
	
	/// Count of bytes to be written 
	cbWriteData			: UDINT;
	
	nOffset			: UDINT;
	nArg			: INT;
	bInputDataError	: BOOL;
	bTest			: BOOL := TRUE;
	bDone			: BOOL;
	bBusy			: BOOL;
	bError			: BOOL;
	nErrorID		: DWORD;
	iState			: INT;
END_VAR
VAR CONSTANT
	nNumberOfInputArguments	: UDINT := 1;
	nNumberOfOutputArguments: UDINT := 1;
	nInputArgSize			: UDINT := 162;
END_VAR

(*
CallInOut1DimParams(	[numberIn1(uInt32),	numberIn2(UInt32)]
						[numberOut1(UInt32),numberOut2(UINT32),	numberOut3(UINT32)]
);
*)

CASE iState OF

0:	(* idle *)
	IF bTest THEN
		bTest		:= FALSE;
		bError		:= FALSE;
		nErrorID	:= 0;
		stOutputArgInfoAndData.sOutArray[1] 	:= ''; 
		stOutputArgInfoAndData.sOutArray[2] 	:= ''; 
		stOutputArgInfoAndData.sOutArray[3] 	:= ''; 
		(* Parameterize *)
		sOpcUA_URL		:= 'opc.tcp://localhost:4841';	(* OpcUA Url of the device with ip address *)

		SessionConnectInfo.tConnectTimeout 		:= T#9M;
		SessionConnectInfo.tSessionTimeout 		:= T#9M;
		SessionConnectInfo.sApplicationName		:= '';
		SessionConnectInfo.sApplicationUri 		:= '';
		SessionConnectInfo.eSecurityMode 		:= eUASecurityMsgMode_None;
		SessionConnectInfo.eSecurityPolicyUri 	:= eUASecurityPolicy_None;
		SessionConnectInfo.eTransportProfileUri := eUATransportProfileUri_UATcp;

		iState	:= iState + 1;
	END_IF

1:	(* open UA session *)
	fbUA_Connect(
		Execute				:= TRUE,
		ServerURL			:= sOpcUA_URL,
		SessionConnectInfo	:= SessionConnectInfo,
		Timeout				:= T#10S,
		ConnectionHdl		=> nConnectionHdl
	);

	IF NOT fbUA_Connect.Busy THEN
		fbUA_Connect(Execute := FALSE);

		IF NOT fbUA_Connect.Error THEN
			(* connected *)
			iState := iState + 1;
		ELSE
			bError			:= TRUE;
			nErrorID		:= fbUA_Connect.ErrorID;
			nConnectionHdl	:= 0;
			iState 			:= 0; (* idle *)
		END_IF
	END_IF


2:	(* GetNS Index *)
	fbUA_GetNamespaceIndex(
		Execute			:= TRUE,
		ConnectionHdl	:= nConnectionHdl,
		NamespaceUri	:= 'PLC1',
		NamespaceIndex	=> nNamespaceIndex
	);

	IF NOT fbUA_GetNamespaceIndex.Busy THEN
		fbUA_GetNamespaceIndex(Execute := FALSE);

		IF NOT fbUA_GetNamespaceIndex.Error THEN
			(* namespace index read successfully *)
			iState 		:= iState + 1; (* get node handle *)
		ELSE
			bError		:= TRUE;
			nErrorID	:= fbUA_GetNamespaceIndex.ErrorID;
			iState 		:= 7; (* disconnect *)
		END_IF
	END_IF

3:	(* Get Method Handle *)
		ObjectNodeID.eIdentifierType := eUAIdentifierType_String;
		ObjectNodeID.nNamespaceIndex := nNamespaceIndex;
		ObjectNodeID.sIdentifier	:= 'TestMethods';
	
		MethodNodeID.eIdentifierType := eUAIdentifierType_String;
		MethodNodeID.nNamespaceIndex := nNamespaceIndex;
		MethodNodeID.sIdentifier	:= 'TestMethods.CallInOut1DimStringParam';

		M_Init();
		IF bInputDataError = FALSE THEN
			iState 	:= iState + 1;
		ELSE
			bBusy		:= FALSE; 
			bError 		:= TRUE;
			nErrorID 	:= 16#70A; //out of memory
		END_IF


4:	(* Method Get Handle *)
	fbUA_MethodGetHandle(
			Execute			:= TRUE,
			ConnectionHdl	:= nConnectionHdl,
			ObjectNodeID	:= ObjectNodeID,
			MethodNodeID 	:= MethodNodeID,
			MethodHdl		=> nMethodHdl
		);
	IF NOT fbUA_MethodGetHandle.Busy THEN
		fbUA_MethodGetHandle(Execute := FALSE);

		IF NOT fbUA_MethodGetHandle.Error THEN
			(*  *)
			iState := iState + 1; (* Call Method *)
		ELSE
			bError		:= TRUE;
			nErrorID	:= fbUA_MethodGetHandle.ErrorID;
			iState	 	:= 6; (* Release method Handle *)
		END_IF
	END_IF


5:	(* Method Call *)
	fbUA_MethodCall(
		Execute					:= TRUE,
		Timeout					:= T#20S,
		ConnectionHdl			:= nConnectionHdl,
		MethodHdl				:= nMethodHdl,
		nNumberOfInputArguments := nNumberOfInputArguments,		(* 1*)
		pInputArgData			:= ADR(nInputData),
		cbInputArgData			:= cbWriteData,
		pInputArgInfo			:= ADR(InputArguments),
		cbInputArgInfo			:= SIZEOF(InputArguments),
		nNumberOfOutputArguments:= nNumberOfOutputArguments,
		pOutputArgInfo			:= ADR(stOutputArgInfo),
		cbOutputArgInfo			:= SIZEOF(stOutputArgInfo),
		pOutputArgInfoAndData	:= ADR(stOutputArgInfoAndData),
		cbOutputArgInfoAndData	:= SIZEOF(stOutputArgInfoAndData)
	);
	IF NOT fbUA_MethodCall.Busy THEN
		fbUA_MethodCall(Execute := FALSE);

		IF NOT fbUA_MethodCall.Error THEN
			(*  *)
			iState 	:= iState + 1; (* Release handle *)
		ELSE
			bError		:= TRUE;
			nErrorID	:= fbUA_MethodCall.ErrorID;
			iState		:= 6; (* Release method handle *)
		END_IF
	END_IF


6:	(* Release Method Handle *)
	fbUA_MethodReleaseHandle(
		Execute			:= TRUE,
		ConnectionHdl	:= nConnectionHdl,
		MethodHdl		:= nMethodHdl
	);

	IF NOT fbUA_MethodReleaseHandle.Busy THEN
		fbUA_MethodReleaseHandle(Execute := FALSE);
		bBusy := FALSE;
		IF NOT fbUA_MethodReleaseHandle.Error THEN
			(* session closed *)
			iState 	:= 7; (* Disconnect *)
		ELSE
			bError		:= TRUE;
			nErrorID	:= fbUA_MethodReleaseHandle.ErrorID;
			iState 		:= 7; (* Disconnect *)
		END_IF
	END_IF
	
7:	(* Disconnect *) 
	fbUA_Disconnect(
		Execute			:= TRUE,
		ConnectionHdl	:= nConnectionHdl
	);

	IF NOT fbUA_Disconnect.Busy THEN
		fbUA_Disconnect(Execute := FALSE);

		IF NOT fbUA_Disconnect.Error THEN
			(* disconnected *)
			iState 			:= 0; (* idle *)
			bDone 	:= TRUE;
			bBusy 	:= FALSE;
		ELSE
			bBusy 	:= FALSE;
			bError			:= TRUE;
			nErrorID		:= fbUA_Disconnect.ErrorID;
			iState 			:= 0; (* idle *)
			nConnectionHdl	:= 0;
		END_IF
	END_IF
END_CASE

ACTION M_Init:
bInputDataError := FALSE; 
nOffset := 0;
MEMSET(ADR(InputArguments),0,SIZEOF(InputArguments));
MEMSET(ADR(nInputData),0,SIZEOF(nInputData));

nArg := 1;
(*numberIn1*)			(********** Input parameter 1 **********)
InputArguments[nArg].DataType			:= eUAType_String;
InputArguments[nArg].ValueRank			:= 1; 							(* Scalar = -1 or 1Dim-Array =1*)
InputArguments[nArg].ArrayDimensions[1]	:= 2; 							(* Number of Dimension in case its an array *)
InputArguments[nArg].nLenData			:= SIZEOF(sInArray);			(* Length if its a STRING *)
IF nOffset + SIZEOF(sInArray) > nInputArgSize THEN 
	bInputDataError := TRUE;
	RETURN;
ELSE
	MEMCPY(ADR(nInputData)+nOffset,ADR(sInArray),SIZEOF(sInArray));			(* VALUE in BYTES FORM *)
	nOffset := nOffset + SIZEOF(sInArray);
END_IF
//InputArguments[nArg].nLenData			:= SIZEOF(sIn1)+SIZEOF(sIn2);			(* Length if its a STRING *)
//MEMCPY(ADR(nInputData)+nOffset,ADR(sIn1),SIZEOF(sIn1));				(* VALUE in BYTES FORM *)
//nOffset := nOffset + SIZEOF(sIn1);
//MEMCPY(ADR(nInputData)+nOffset,ADR(sIn2),SIZEOF(sIn2));				(* VALUE in BYTES FORM *)
//nOffset := nOffset + SIZEOF(sIn2);

cbWriteData := nOffset;

// ************* Prepare Output variable info **************
stOutputArgInfo[1].nLenData := SIZEOF(stOutputArgInfoAndData.sOutArray);
END_ACTION

END_PROGRAM

// ---- Tests_Henning/POUs/PRG_CallInOutMultiParam.TcPOU
PROGRAM PRG_CallInOutMultiParam
VAR
	///CallInOutMultiParams(numberIn1(uInt32),numberIn2(UInt32),numberOut1(UInt32),numberOut2(UINT32));
	fbUA_Connect			: UA_Connect;
	SessionConnectInfo		: ST_UASessionConnectInfo;
	sOpcUA_URL				: STRING(MAX_STRING_LENGTH);
	nConnectionHdl			: DWORD;
	
	fbUA_GetNamespaceIndex	: UA_GetNamespaceIndex;
	nNamespaceIndex			: UINT;

	fbUA_MethodGetHandle: UA_MethodGetHandle;
	nMethodHdl			: DWORD;
	ObjectNodeID		: ST_UANodeID;
	MethodNodeID		: ST_UANodeID;
	
	fbUA_MethodCall		: UA_MethodCall;
	InputArguments		: ARRAY[1..nNumberOfInputArguments] OF ST_UAMethodArgInfo;
	nInputData			: ARRAY[1..nInputArgSize] OF BYTE;
	OutputArgAndData	: ST_UAMethodCall_CallInOutParam;
	stOutputArgInfo		: ARRAY [1..nNumberOfOutputArguments] OF ST_UAMethodArgInfo;
	
	numberIn1		: UDINT;
	numberIn2		: UDINT;
		
	fbUA_MethodReleaseHandle	: UA_MethodReleaseHandle;
	
	fbUA_Disconnect	: UA_Disconnect;
	
	nArg			: INT;
	cbWriteData		: UDINT;
	nOffset			: UDINT;
	bInputDataError	: BOOL;
	
	bTest		: BOOL := TRUE;
	bDone		: BOOL;
	bBusy		: BOOL;
	bError		: BOOL;
	nErrorID	: DWORD;
	iState		: INT;
END_VAR
VAR CONSTANT
	nNumberOfInputArguments	: UDINT := 2;
	nNumberOfOutputArguments: UDINT := 2; 
	nInputArgSize			: UDINT := 8; 
END_VAR

(*
CallInOutMultiParams(	numberIn1(uInt32),
						numberIn2(UInt32),
						numberOut1(UInt32),
						numberOut2(UINT32)	);
*)

CASE iState OF

0:	(* idle *)
	IF bTest THEN
		bTest		:= FALSE;
		bError		:= FALSE;
		nErrorID	:= 0;
		OutputArgAndData.output1 	:= 0; 
		OutputArgAndData.output2 	:= 0; 
		(* Parameterize *)
		sOpcUA_URL		:= 'opc.tcp://localhost:4841';	(* OpcUA Url of the device with ip address *)

		SessionConnectInfo.tConnectTimeout 		:= T#9S;
		SessionConnectInfo.tSessionTimeout 		:= T#9S;
		SessionConnectInfo.sApplicationName		:= '';
		SessionConnectInfo.sApplicationUri 		:= '';
		SessionConnectInfo.eSecurityMode 		:= eUASecurityMsgMode_None;
		SessionConnectInfo.eSecurityPolicyUri 	:= eUASecurityPolicy_None;
		SessionConnectInfo.eTransportProfileUri := eUATransportProfileUri_UATcp;

		iState	:= iState + 1;
	END_IF

1:	(* open UA session *)
	fbUA_Connect(
		Execute				:= TRUE,
		ServerURL			:= sOpcUA_URL,
		SessionConnectInfo	:= SessionConnectInfo,
		Timeout				:= T#10S,
		ConnectionHdl		=> nConnectionHdl
	);

	IF NOT fbUA_Connect.Busy THEN
		fbUA_Connect(Execute := FALSE);

		IF NOT fbUA_Connect.Error THEN
			(* connected *)
			iState := iState + 1;
		ELSE
			bError			:= TRUE;
			nErrorID		:= fbUA_Connect.ErrorID;
			nConnectionHdl	:= 0;
			iState 			:= 0; (* idle *)
		END_IF
	END_IF


2:	(* GetNS Index *)
	fbUA_GetNamespaceIndex(
		Execute			:= TRUE,
		ConnectionHdl	:= nConnectionHdl,
		NamespaceUri	:= 'PLC1',
		NamespaceIndex	=> nNamespaceIndex
	);

	IF NOT fbUA_GetNamespaceIndex.Busy THEN
		fbUA_GetNamespaceIndex(Execute := FALSE);

		IF NOT fbUA_GetNamespaceIndex.Error THEN
			(* namespace index read successfully *)
			iState 		:= iState + 1; (* get node handle *)
		ELSE
			bError		:= TRUE;
			nErrorID	:= fbUA_GetNamespaceIndex.ErrorID;
			iState 		:= 7; (* disconnect *)
		END_IF
	END_IF

3:	(* Get Method Handle *)
		ObjectNodeID.eIdentifierType := eUAIdentifierType_String;
		ObjectNodeID.nNamespaceIndex := nNamespaceIndex;
		ObjectNodeID.sIdentifier	:= 'TestMethods';
	
		MethodNodeID.eIdentifierType := eUAIdentifierType_String;
		MethodNodeID.nNamespaceIndex := nNamespaceIndex;
		MethodNodeID.sIdentifier	:= 'TestMethods.CallInOutMultiParams';

		M_Init();
		IF bInputDataError = FALSE THEN
			iState 	:= iState + 1;
		ELSE
			bBusy		:= FALSE; 
			bError 		:= TRUE;
			nErrorID 	:= 16#70A; //out of memory
		END_IF


4:	(* Method Get Handle *)
	fbUA_MethodGetHandle(
			Execute			:= TRUE,
			ConnectionHdl	:= nConnectionHdl,
			ObjectNodeID	:= ObjectNodeID,
			MethodNodeID 	:= MethodNodeID,
			MethodHdl		=> nMethodHdl
		);
	IF NOT fbUA_MethodGetHandle.Busy THEN
		fbUA_MethodGetHandle(Execute := FALSE);

		IF NOT fbUA_MethodGetHandle.Error THEN
			(*  *)
			iState := iState + 1; (* Call Method *)
		ELSE
			bError		:= TRUE;
			nErrorID	:= fbUA_MethodGetHandle.ErrorID;
			iState	 	:= 6; (* Release method Handle *)
		END_IF
	END_IF


5:	(* Method Call *)	
	fbUA_MethodCall(
		Execute					:= TRUE,
		Timeout					:= T#20S,
		ConnectionHdl			:= nConnectionHdl,
		MethodHdl				:= nMethodHdl,
		nNumberOfInputArguments := nNumberOfInputArguments,		(* 2 *)
		pInputArgData			:= ADR(nInputData),
		cbInputArgData			:= cbWriteData,
		pInputArgInfo			:= ADR(InputArguments),
		cbInputArgInfo			:= SIZEOF(InputArguments),
		nNumberOfOutputArguments:= nNumberOfOutputArguments,		(* 2 *)
		pOutputArgInfo 			:= ADR(stOutputArgInfo),
		cbOutputArgInfo			:= SIZEOF(stOutputArgInfo),
		pOutputArgInfoAndData	:= ADR(OutputArgAndData),
		cbOutputArgInfoAndData	:= SIZEOF(OutputArgAndData)
	);
	IF NOT fbUA_MethodCall.Busy THEN
		fbUA_MethodCall(Execute := FALSE);

		IF NOT fbUA_MethodCall.Error THEN
			(*  *)
			iState 	:= iState + 1; (* Release handle *)
			//MEMCPY(ADR(OutputArgAndData.output1),ADR(OutputArguments),SIZEOF(OutputArgAndData.output1));
			//MEMCPY(ADR(OutputArgAndData.output2),ADR(OutputArguments)+SIZEOF(OutputArgAndData.output1),SIZEOF(OutputArgAndData.output2));
		ELSE
			bError		:= TRUE;
			nErrorID	:= fbUA_MethodCall.ErrorID;
			iState		:= 6; (* Release method handle *)
		END_IF
	END_IF


6:	(* Release Method Handle *)
	fbUA_MethodReleaseHandle(
		Execute			:= TRUE,
		ConnectionHdl	:= nConnectionHdl,
		MethodHdl		:= nMethodHdl
	);

	IF NOT fbUA_MethodReleaseHandle.Busy THEN
		fbUA_MethodReleaseHandle(Execute := FALSE);
		bBusy := FALSE;
		IF NOT fbUA_MethodReleaseHandle.Error THEN
			(* session closed *)
			iState 	:= 7; (* Disconnect *)
		ELSE
			bError		:= TRUE;
			nErrorID	:= fbUA_MethodReleaseHandle.ErrorID;
			iState 		:= 7; (* Disconnect *)
		END_IF
	END_IF
	
7:	(* Disconnect *) 
	fbUA_Disconnect(
		Execute			:= TRUE,
		ConnectionHdl	:= nConnectionHdl
	);

	IF NOT fbUA_Disconnect.Busy THEN
		fbUA_Disconnect(Execute := FALSE);

		IF NOT fbUA_Disconnect.Error THEN
			(* disconnected *)
			iState 			:= 0; (* idle *)
			bDone 	:= TRUE;
			bBusy 	:= FALSE;
		ELSE
			bBusy 	:= FALSE;
			bError			:= TRUE;
			nErrorID		:= fbUA_Disconnect.ErrorID;
			iState 			:= 0; (* idle *)
			nConnectionHdl	:= 0;
		END_IF
	END_IF
END_CASE

ACTION M_Init:
bInputDataError := FALSE; 
nOffset := 0;
MEMSET(ADR(InputArguments),0,SIZEOF(InputArguments));
MEMSET(ADR(nInputData),0,SIZEOF(nInputData));

nArg := 1;
(*numberIn1*)			(********** Input parameter 1 **********)
InputArguments[nArg].DataType			:= eUAType_UInt32;
InputArguments[nArg].ValueRank			:= -1; 							(* Scalar = -1 or Array *)
InputArguments[nArg].ArrayDimensions[1]	:= 0; 							(* Number of Dimension in case its an array *)
InputArguments[nArg].nLenData			:= SIZEOF(numberIn1);			(* Length if its a STRING *)
IF nOffset + SIZEOF(numberIn1) > nInputArgSize THEN 
	bInputDataError := TRUE;
	RETURN;
ELSE
	MEMCPY(ADR(nInputData)+nOffset,ADR(numberIn1),SIZEOF(numberIn1));				(* VALUE in BYTES FORM *)
	nOffset := nOffset + SIZEOF(numberIn1);
END_IF

cbWriteData := nOffset;
nArg := nArg + 1;
(* numberIn2;*)			(********** Input parameter 2 **********)
InputArguments[nArg].DataType			:= eUAType_UInt32;
InputArguments[nArg].ValueRank			:= -1; 							(* Scalar = -1 or Array *)
InputArguments[nArg].ArrayDimensions[1]	:= 0; 							(* Number of Dimension in case its an array *)
InputArguments[nArg].nLenData			:= SIZEOF(numberIn2);				(* Length if its a STRING *)
IF nOffset + SIZEOF(numberIn2) > nInputArgSize THEN 
	bInputDataError := TRUE;
	RETURN;
ELSE
	MEMCPY(ADR(nInputData)+nOffset,ADR(numberIn2),SIZEOF(numberIn2));				(* VALUE in BYTES FORM *)
	nOffset := nOffset + SIZEOF(numberIn2);
END_IF

cbWriteData := nOffset;

// ************* Prepare Output variable info **************
stOutputArgInfo[1].nLenData := SIZEOF(OutputArgAndData.output1);
stOutputArgInfo[2].nLenData := SIZEOF(OutputArgAndData.output2);
END_ACTION

END_PROGRAM

// ---- Tests_Henning/POUs/PRG_ScalarTest.TcPOU
PROGRAM PRG_ScalarTest
VAR
	iState: INT;
END_VAR

CASE iState OF
0:	
	PRG_ScalarTest_Read();
	IF(NOT PRG_ScalarTest_Read.bBusy AND NOT PRG_ScalarTest_Read.bError) THEN
		iState := iState+1;
		//Reset thus could be reused
		//PRG_ScalarTest_Read.nLoopVars := 0;
		//PRG_ScalarTest_Read.nLoopVars := 0;
	END_IF
1:
	PRG_ScalarTest_Write();
	IF(NOT PRG_ScalarTest_Write.bBusy AND NOT PRG_ScalarTest_Write.bError) THEN
		iState := iState+1;
	END_IF
2:
	PRG_ScalarTest_ReadWritten();
	IF(NOT PRG_ScalarTest_ReadWritten.bBusy AND NOT PRG_ScalarTest_ReadWritten.bError) THEN
		iState := iState+1;
	END_IF
END_CASE

END_PROGRAM

// ---- Tests_Henning/POUs/PRG_ScalarTest_Read.TcPOU
PROGRAM PRG_ScalarTest_Read
VAR
	fbUA_Connect: UA_Connect;
	SessionConnectInfo: ST_UASessionConnectInfo;
	nConnectionHdl: DWORD;
	fbUA_GetNamespaceIndex: UA_GetNamespaceIndex;
	nNamespaceIndex: UINT;
	fbUA_NodeGetHandle: UA_NodeGetHandle;
	NodeID: ST_UANodeID;
	nNodeHdl: DWORD;
	fbUA_Read: UA_Read;
	stIndexRange: ARRAY[1..nMaxIndexRange] OF ST_UAIndexRange;
	nIndexRangeCount: UINT;
	stNodeAddInfo: ST_UANodeAdditionalInfo;
	Variable: ARRAY[1..nMaxReadData] OF BYTE;
	///DINT; 		// change the data type according to the variable type to be read
	nReadData: STRING;
	fbUA_NodeReleaseHandle: UA_NodeReleaseHandle;
	fbUA_Disconnect: UA_Disconnect;
	iState: INT;
	bTest: BOOL := TRUE;
	bDone: BOOL;
	bBusy: BOOL;
	bError: BOOL;
	nErrorID: DWORD;
	nLoopVars: UINT;
END_VAR

CASE iState OF
0:	(* idle *)
	IF bTest THEN
		bTest		:= FALSE;
		bError		:= FALSE;
		nErrorID	:= 0;
		bBusy 		:= TRUE; 
		SessionConnectInfo.tConnectTimeout 		:= T#9S;
		SessionConnectInfo.tSessionTimeout 		:= T#9S;
		SessionConnectInfo.sApplicationName		:= '';
		SessionConnectInfo.sApplicationUri 		:= '';
		SessionConnectInfo.eSecurityMode 		:= eUASecurityMsgMode_None;
		SessionConnectInfo.eSecurityPolicyUri 	:= eUASecurityPolicy_None;
		SessionConnectInfo.eTransportProfileUri := eUATransportProfileUri_UATcp;

		stNodeAddInfo.nIndexRangeCount := nIndexRangeCount;
		stNodeAddInfo.stIndexRange := stIndexRange;
		iState	:= iState + 1;
	END_IF

1:	(* open UA session *)
	fbUA_Connect(
		Execute				:= TRUE,
		ServerURL			:= GVL_ScalarTests.sOpcUA_URL,
		SessionConnectInfo	:= SessionConnectInfo,
		Timeout				:= T#10S,
		ConnectionHdl		=> nConnectionHdl
	);

	IF NOT fbUA_Connect.Busy THEN
		fbUA_Connect(Execute := FALSE);

		IF NOT fbUA_Connect.Error THEN
			(* session open *)
			iState := iState + 1;
		ELSE
			bError			:= TRUE;
			nErrorID		:= fbUA_Connect.ErrorID;
			nConnectionHdl	:= 0;
			iState 			:= 0; (* idle *)
		END_IF
	END_IF


2:	(* GetNS Index *)
	fbUA_GetNamespaceIndex(
		Execute			:= TRUE,
		ConnectionHdl	:= nConnectionHdl,
		NamespaceUri	:= GVL_ScalarTests.sNodeIDNamespace,
		NamespaceIndex	=> nNamespaceIndex
	);

	IF NOT fbUA_GetNamespaceIndex.Busy THEN
		fbUA_GetNamespaceIndex(Execute := FALSE);

		IF NOT fbUA_GetNamespaceIndex.Error THEN
			(* session closed *)
			iState 		:= iState + 1; (* idle *)
		ELSE
			bError		:= TRUE;
			nErrorID	:= fbUA_GetNamespaceIndex.ErrorID;
			iState 		:= 6; (* idle *)
		END_IF
	END_IF


3:	(* Get Node Handle *)
	NodeID.eIdentifierType := eUAIdentifierType_String;
	NodeID.nNamespaceIndex := nNamespaceIndex;
	NodeID.sIdentifier	:= GVL_ScalarTests.NodeID_Identifiers[nLoopVars]; // 'GVL_static.stat_BSTR_0';
	fbUA_NodeGetHandle(
		Execute			:= TRUE,
		ConnectionHdl	:= nConnectionHdl,
		NodeID			:= NodeID,
		NodeHdl			=> nNodeHdl
	);

	IF NOT fbUA_NodeGetHandle.Busy THEN
		fbUA_NodeGetHandle(Execute := FALSE);

		IF NOT fbUA_NodeGetHandle.Error THEN
			(* session closed *)
			iState 		:= iState + 1; (* idle *)
		ELSE
			bError		:= TRUE;
			nErrorID	:= fbUA_NodeGetHandle.ErrorID;
			iState 		:= 6; (* idle *)
		END_IF
	END_IF


4: 	(* UA_Read *)
	fbUA_Read(
		Execute			:= TRUE,
		ConnectionHdl	:= nConnectionHdl,
		NodeHdl			:= nNodeHdl,
		stNodeAddInfo 	:= stNodeAddInfo,
		cbData			:= GVL_ScalarTests.NodeID_Sizes[nLoopVars], //SIZEOF(nReadData),
		pVariable		:= ADR(GVL_ScalarTests.NodeID_ReadResults[nLoopVars].nData) //Variable
		);

	IF NOT fbUA_Read.Busy THEN
		fbUA_Read(
			Execute 	:= FALSE);

		IF NOT fbUA_Read.Error THEN
			(* session closed *)
			iState 		:= iState + 1; (* idle *)
			//Do we need this? We simply store in UNION! MEMCPY(ADR(nReadData),ADR(Variable),SIZEOF(nReadData));
		ELSE
			bError		:= TRUE;
			nErrorID	:= fbUA_Read.ErrorID;
			iState 		:= 6; (* idle *)
		END_IF
	END_IF



5:	(* Release Node Handle *)
	fbUA_NodeReleaseHandle(
		Execute			:= TRUE,
		ConnectionHdl	:= nConnectionHdl,
		NodeHdl			:= nNodeHdl
	);

	IF NOT fbUA_NodeReleaseHandle.Busy THEN
		fbUA_NodeReleaseHandle(Execute := FALSE);

		IF NOT fbUA_NodeReleaseHandle.Error THEN
			(* session closed *)
			iState 		:= iState + 1; (* idle *)
		ELSE
			bError		:= TRUE;
			nErrorID	:= fbUA_NodeReleaseHandle.ErrorID;
			iState 		:= 6; (* idle *)
		END_IF
	END_IF


6:	(* close session *)
	fbUA_Disconnect(
		Execute			:= TRUE,
		ConnectionHdl	:= nConnectionHdl
	);

	IF NOT fbUA_Disconnect.Busy THEN
		fbUA_Disconnect(Execute := FALSE);

		IF NOT fbUA_Disconnect.Error THEN
			(* session closed *)
			iState 		:= 0; (* idle *)
			//restart with next var, if existing in array
			IF(nLoopVars < nEndOfNodeIDVars) THEN
				nLoopVars := nLoopVars+1;
				bTest := TRUE;
			ELSE 
				bBusy 		:= FALSE;
				//prepare for next call 
				bTest := TRUE;
				nLoopVars := 0;
			END_IF
		ELSE
			bError			:= TRUE;
			nErrorID		:= fbUA_Disconnect.ErrorID;
			iState 			:= 0; (* idle *)
			nConnectionHdl	:= 0;
		END_IF
	END_IF
END_CASE

END_PROGRAM

// ---- Tests_Henning/POUs/PRG_ScalarTest_Write.TcPOU
PROGRAM PRG_ScalarTest_Write
VAR
	fbUA_Connect: UA_Connect;
	SessionConnectInfo: ST_UASessionConnectInfo;
	sOpcUA_URL: STRING(MAX_STRING_LENGTH);
	nConnectionHdl: DWORD;
	fbUA_GetNamespaceIndex: UA_GetNamespaceIndex;
	sNamespaceUri: STRING(MAX_STRING_LENGTH);
	nNamespaceIndex: UINT;
	fbUA_NodeGetHandle: UA_NodeGetHandle;
	NodeID: ST_UANodeID;
	nNodeHdl: DWORD;
	fbUA_Write: UA_Write;
	stIndexRange: ARRAY[1..nMaxIndexRange] OF ST_UAIndexRange;
	nIndexRangeCount: UINT;
	stNodeAddInfo: ST_UANodeAdditionalInfo;
	/// UDINT := 12312345;		// change according to the type of variable
	nWriteData: STRING := 'Hallo';
	Variable: ARRAY[1..nMaxReadData] OF BYTE;
	cbData: UDINT;
	fbUA_NodeReleaseHandle: UA_NodeReleaseHandle;
	fbUA_Disconnect: UA_Disconnect;
	iState: INT;
	bTest: BOOL := TRUE;
	bDone: BOOL;
	bBusy: BOOL;
	bError: BOOL;
	nErrorID: DWORD;
	nLoopVars: UINT;
END_VAR

CASE iState OF
0:	(* idle *)
	IF bTest THEN
		bTest	:= FALSE;
		bError	:= FALSE;
		nErrorID	:= 0;
		bBusy := TRUE; 

		(* Parameterize 
		GVL_ScalarTests.NodeID_WriteCommands[0].bBool := TRUE; 
		GVL_ScalarTests.NodeID_WriteCommands[1].sString := 'WriteTest'; 
		GVL_ScalarTests.NodeID_WriteCommands[2].bByte := 123; 
		GVL_ScalarTests.NodeID_WriteCommands[3].nInt := 124; 
		GVL_ScalarTests.NodeID_WriteCommands[4].nUdint := 125; 
		GVL_ScalarTests.NodeID_WriteCommands[5].nLReal := 1.23456; //R8x 
		GVL_ScalarTests.NodeID_WriteCommands[6].bByte := 111; 
		GVL_ScalarTests.NodeID_WriteCommands[7].nInt := 112; 
		GVL_ScalarTests.NodeID_WriteCommands[8].nUdint := 113; 
		*)
		
		
		
		SessionConnectInfo.tConnectTimeout 		:= T#9S;
		SessionConnectInfo.tSessionTimeout 		:= T#9S;
		SessionConnectInfo.sApplicationName		:= '';
		SessionConnectInfo.sApplicationUri 		:= '';
		SessionConnectInfo.eSecurityMode 		:= eUASecurityMsgMode_None;
		SessionConnectInfo.eSecurityPolicyUri 	:= eUASecurityPolicy_None;
		SessionConnectInfo.eTransportProfileUri := eUATransportProfileUri_UATcp;
		
		stNodeAddInfo.nIndexRangeCount := nIndexRangeCount;
		stNodeAddInfo.stIndexRange := stIndexRange;
		iState	:= iState + 1;
	END_IF

1:	(* open UA session *)
	fbUA_Connect(
		Execute				:= TRUE,
		ServerURL			:= GVL_ScalarTests.sOpcUA_URL,
		SessionConnectInfo	:= SessionConnectInfo,
		Timeout				:= T#10S,
		ConnectionHdl		=> nConnectionHdl
	);

	IF NOT fbUA_Connect.Busy THEN
		fbUA_Connect(Execute := FALSE);

		IF NOT fbUA_Connect.Error THEN
			(* session open *)
			iState := iState + 1;
		ELSE
			bError			:= TRUE;
			nErrorID		:= fbUA_Connect.ErrorID;
			nConnectionHdl	:= 0;
			iState 			:= 0; (* idle *)
		END_IF
	END_IF


2:	(* GetNS Index *)
	fbUA_GetNamespaceIndex(
		Execute			:= TRUE,
		ConnectionHdl	:= nConnectionHdl,
		NamespaceUri	:= GVL_ScalarTests.sNodeIDNamespace,
		NamespaceIndex	=> nNamespaceIndex
	);

	IF NOT fbUA_GetNamespaceIndex.Busy THEN
		fbUA_GetNamespaceIndex(Execute := FALSE);

		IF NOT fbUA_GetNamespaceIndex.Error THEN
			(* session closed *)
			iState 		:= iState + 1; (* idle *)
		ELSE
			bError		:= TRUE;
			nErrorID	:= fbUA_GetNamespaceIndex.ErrorID;
			iState 		:= 6; (* idle *)
		END_IF
	END_IF


3:	(* Get Node Handle *)
	NodeID.eIdentifierType := eUAIdentifierType_String;
	NodeID.nNamespaceIndex := nNamespaceIndex;
	NodeID.sIdentifier	:= GVL_ScalarTests.NodeID_Identifiers[nLoopVars]; // 'GVL_static.stat_BSTR_0';
	fbUA_NodeGetHandle(
		Execute			:= TRUE,
		ConnectionHdl	:= nConnectionHdl,
		NodeID			:= NodeID,
		NodeHdl			=> nNodeHdl
	);

	IF NOT fbUA_NodeGetHandle.Busy THEN
		fbUA_NodeGetHandle(Execute := FALSE);

		IF NOT fbUA_NodeGetHandle.Error THEN
			(* session closed *)
			IF SIZEOF(nWriteData) <= nMaxReadData THEN 
				iState 		:= iState + 1; (* idle *)
				MEMSET(ADR(Variable),0,SIZEOF(Variable));
				MEMCPY(ADR(Variable),ADR(nWriteData),SIZEOF(nWriteData));
			ELSE
				//cannot write buffer too small -> increase the value of nMaxData in GVL
				bError		:= TRUE;
				iState 		:= 6; (* idle *)
			END_IF
		ELSE
			bError		:= TRUE;
			nErrorID	:= fbUA_NodeGetHandle.ErrorID;
			iState 		:= 6; (* idle *)
		END_IF
	END_IF


4: 	(* UA_Write *)
	fbUA_Write(
		Execute			:= TRUE,
		ConnectionHdl	:= nConnectionHdl,
		NodeHdl			:= nNodeHdl,
		stNodeAddInfo	:= stNodeAddInfo,
		cbData			:= GVL_ScalarTests.NodeID_Sizes[nLoopVars], //SIZEOF(nWriteData),
		pVariable		:= ADR(GVL_ScalarTests.NodeID_WriteCommands[nLoopVars].nData) // Variable		:= Variable
		);

	IF NOT fbUA_Write.Busy THEN
		fbUA_Write(
			Execute 		:= FALSE);

		IF NOT fbUA_Write.Error THEN
			(* session closed *)
			iState 		:= iState + 1; (* idle *)
		ELSE
			bError		:= TRUE;
			nErrorID	:= fbUA_Write.ErrorID;
			iState 		:= 6; (* idle *)
		END_IF
	END_IF


5:	(* Release Node Handle *)
	fbUA_NodeReleaseHandle(
		Execute			:= TRUE,
		ConnectionHdl	:= nConnectionHdl,
		NodeHdl			:= nNodeHdl
	);

	IF NOT fbUA_NodeReleaseHandle.Busy THEN
		fbUA_NodeReleaseHandle(Execute := FALSE);

		IF NOT fbUA_NodeReleaseHandle.Error THEN
			(* session closed *)
			iState 		:= iState + 1; (* idle *)
		ELSE
			bError		:= TRUE;
			nErrorID	:= fbUA_NodeReleaseHandle.ErrorID;
			iState 		:= 6; (* idle *)
		END_IF
	END_IF


6:	(* close session *)
	fbUA_Disconnect(
		Execute			:= TRUE,
		ConnectionHdl	:= nConnectionHdl
	);

	IF NOT fbUA_Disconnect.Busy THEN
		fbUA_Disconnect(Execute := FALSE);

		IF NOT fbUA_Disconnect.Error THEN
			(* session closed *)
			iState 		:= 0; (* idle *)			//restart with next var, if existing in array
			IF(nLoopVars < nEndOfNodeIDVars) THEN
				nLoopVars := nLoopVars+1;
				bTest := TRUE;
			ELSE 
				bBusy 		:= FALSE;
				//prepare for next call 
				nLoopVars := 0;
			END_IF
		ELSE
			bError		:= TRUE;
			nErrorID	:= fbUA_Disconnect.ErrorID;
			iState 		:= 0; (* idle *)
			nConnectionHdl	:= 0;
		END_IF
	END_IF
END_CASE

END_PROGRAM

// ---- Tests_Henning/POUs/PRG_ScalarTest_ReadWritten.TcPOU
PROGRAM PRG_ScalarTest_ReadWritten
VAR
	fbUA_Connect: UA_Connect;
	SessionConnectInfo: ST_UASessionConnectInfo;
	nConnectionHdl: DWORD;
	fbUA_GetNamespaceIndex: UA_GetNamespaceIndex;
	nNamespaceIndex: UINT;
	fbUA_NodeGetHandle: UA_NodeGetHandle;
	NodeID: ST_UANodeID;
	nNodeHdl: DWORD;
	fbUA_Read: UA_Read;
	stIndexRange: ARRAY[1..nMaxIndexRange] OF ST_UAIndexRange;
	nIndexRangeCount: UINT;
	stNodeAddInfo: ST_UANodeAdditionalInfo;
	Variable: ARRAY[1..nMaxReadData] OF BYTE;
	///DINT; 		// change the data type according to the variable type to be read
	nReadData: STRING;
	fbUA_NodeReleaseHandle: UA_NodeReleaseHandle;
	fbUA_Disconnect: UA_Disconnect;
	iState: INT;
	bTest: BOOL := TRUE;
	bDone: BOOL;
	bBusy: BOOL;
	bError: BOOL;
	nErrorID: DWORD;
	nLoopVars: UINT;
	counter: UDINT;
	a: ARRAY[1..nMaxReadData] OF BYTE;
	b: ARRAY[1..nMaxReadData] OF BYTE;
	a_: BYTE;
	b_: BYTE;
END_VAR

CASE iState OF
0:	(* idle *)
	IF bTest THEN
		bTest		:= FALSE;
		bError		:= FALSE;
		nErrorID	:= 0;
		bBusy 		:= TRUE; 
		SessionConnectInfo.tConnectTimeout 		:= T#9S;
		SessionConnectInfo.tSessionTimeout 		:= T#9S;
		SessionConnectInfo.sApplicationName		:= '';
		SessionConnectInfo.sApplicationUri 		:= '';
		SessionConnectInfo.eSecurityMode 		:= eUASecurityMsgMode_None;
		SessionConnectInfo.eSecurityPolicyUri 	:= eUASecurityPolicy_None;
		SessionConnectInfo.eTransportProfileUri := eUATransportProfileUri_UATcp;

		stNodeAddInfo.nIndexRangeCount := nIndexRangeCount;
		stNodeAddInfo.stIndexRange := stIndexRange;
		iState	:= iState + 1;
	END_IF

1:	(* open UA session *)
	fbUA_Connect(
		Execute				:= TRUE,
		ServerURL			:= GVL_ScalarTests.sOpcUA_URL,
		SessionConnectInfo	:= SessionConnectInfo,
		Timeout				:= T#10S,
		ConnectionHdl		=> nConnectionHdl
	);

	IF NOT fbUA_Connect.Busy THEN
		fbUA_Connect(Execute := FALSE);

		IF NOT fbUA_Connect.Error THEN
			(* session open *)
			iState := iState + 1;
		ELSE
			bError			:= TRUE;
			nErrorID		:= fbUA_Connect.ErrorID;
			nConnectionHdl	:= 0;
			iState 			:= 0; (* idle *)
		END_IF
	END_IF


2:	(* GetNS Index *)
	fbUA_GetNamespaceIndex(
		Execute			:= TRUE,
		ConnectionHdl	:= nConnectionHdl,
		NamespaceUri	:= GVL_ScalarTests.sNodeIDNamespace,
		NamespaceIndex	=> nNamespaceIndex
	);

	IF NOT fbUA_GetNamespaceIndex.Busy THEN
		fbUA_GetNamespaceIndex(Execute := FALSE);

		IF NOT fbUA_GetNamespaceIndex.Error THEN
			(* session closed *)
			iState 		:= iState + 1; (* idle *)
		ELSE
			bError		:= TRUE;
			nErrorID	:= fbUA_GetNamespaceIndex.ErrorID;
			iState 		:= 6; (* idle *)
		END_IF
	END_IF


3:	(* Get Node Handle *)
	NodeID.eIdentifierType := eUAIdentifierType_String;
	NodeID.nNamespaceIndex := nNamespaceIndex;
	NodeID.sIdentifier	:= GVL_ScalarTests.NodeID_Identifiers[nLoopVars]; // 'GVL_static.stat_BSTR_0';
	fbUA_NodeGetHandle(
		Execute			:= TRUE,
		ConnectionHdl	:= nConnectionHdl,
		NodeID			:= NodeID,
		NodeHdl			=> nNodeHdl
	);

	IF NOT fbUA_NodeGetHandle.Busy THEN
		fbUA_NodeGetHandle(Execute := FALSE);

		IF NOT fbUA_NodeGetHandle.Error THEN
			(* session closed *)
			iState 		:= iState + 1; (* idle *)
		ELSE
			bError		:= TRUE;
			nErrorID	:= fbUA_NodeGetHandle.ErrorID;
			iState 		:= 6; (* idle *)
		END_IF
	END_IF


4: 	(* UA_Read *)
	fbUA_Read(
		Execute			:= TRUE,
		ConnectionHdl	:= nConnectionHdl,
		NodeHdl			:= nNodeHdl,
		stNodeAddInfo 	:= stNodeAddInfo,
		cbData			:= GVL_ScalarTests.NodeID_Sizes[nLoopVars], //SIZEOF(nReadData),		
		pVariable		:= ADR(GVL_ScalarTests.NodeID_ReadWrittenResults[nLoopVars].nData) //Variable
		);

	IF NOT fbUA_Read.Busy THEN
		fbUA_Read(
			Execute 	:= FALSE);

		IF NOT fbUA_Read.Error THEN
			(* session closed *)
			iState 		:= iState + 1; (* idle *)
			a := GVL_ScalarTests.NodeID_WriteCommands[nLoopVars].nData;
			b := GVL_ScalarTests.NodeID_ReadWrittenResults[nLoopVars].nData;
			FOR counter:=1 TO fbUA_Read.cbData_R //fbUA_Read.GVL_ScalarTests.NodeID_Sizes[nLoopVars]
			DO
				a_ := a[counter];
				b_ := b[counter];
				IF(NOT a_ = b_) THEN
					EXIT;
				END_IF
			END_FOR
			IF(Counter = fbUA_Read.cbData_R+1) THEN //GVL_ScalarTests.NodeID_Sizes[nLoopVars]+1) THEN //all bytes are equal as long as length site is defined
				GVL_ScalarTests.NodeID_CheckReadWrite[nLoopVars] := TRUE;
			END_IF 
			//Do we need this? We simply store in UNION! MEMCPY(ADR(nReadData),ADR(Variable),SIZEOF(nReadData));
		ELSE
			bError		:= TRUE;
			nErrorID	:= fbUA_Read.ErrorID;
			iState 		:= 6; (* idle *)
		END_IF
	END_IF



5:	(* Release Node Handle *)
	fbUA_NodeReleaseHandle(
		Execute			:= TRUE,
		ConnectionHdl	:= nConnectionHdl,
		NodeHdl			:= nNodeHdl
	);

	IF NOT fbUA_NodeReleaseHandle.Busy THEN
		fbUA_NodeReleaseHandle(Execute := FALSE);

		IF NOT fbUA_NodeReleaseHandle.Error THEN
			(* session closed *)
			iState 		:= iState + 1; (* idle *)
		ELSE
			bError		:= TRUE;
			nErrorID	:= fbUA_NodeReleaseHandle.ErrorID;
			iState 		:= 6; (* idle *)
		END_IF
	END_IF


6:	(* close session *)
	fbUA_Disconnect(
		Execute			:= TRUE,
		ConnectionHdl	:= nConnectionHdl
	);

	IF NOT fbUA_Disconnect.Busy THEN
		fbUA_Disconnect(Execute := FALSE);

		IF NOT fbUA_Disconnect.Error THEN
			(* session closed *)
			iState 		:= 0; (* idle *)
			//restart with next var, if existing in array
			IF(nLoopVars < nEndOfNodeIDVars) THEN
				nLoopVars := nLoopVars+1;
				bTest := TRUE;
			ELSE 
				bBusy 		:= FALSE;
				//prepare for next call 
				bTest := TRUE;
				nLoopVars := 0;
			END_IF
		ELSE
			bError			:= TRUE;
			nErrorID		:= fbUA_Disconnect.ErrorID;
			iState 			:= 0; (* idle *)
			nConnectionHdl	:= 0;
		END_IF
	END_IF
END_CASE

END_PROGRAM
